14: (*химическая дезинфекция*)
Chemical(
	i_Diag:= i_DiagChemicDesinfection ,
	i_Pause:= i_Pause ,
	i_Block_Q4_in:= i_Block_Q4_in_level ,
	i_Alarm_LSmin:= i_Alarm_LSmin_Dez ,
	i_Ready_Route:= i_Ready_Route ,
	i_FS:= i_FS ,
	i_LSL:= i_LSL ,
	i_LSM:= i_LSM ,
	i_LSH:= i_LSH ,
	i_TE1:= i_TE1 ,
	i_TE2:= i_TE2 ,
	i_Current_VolumeFC1:= Current_VolumeFC1 ,
	i_Current_VolumeFC11:= Current_VolumeFC11 ,
	i_TimeDelay:= i_TimeDelay ,
	i_Time_LSH_on:= i_Time_LSH_on ,
	i_Time_LSM_on:= i_Time_LSM_on ,
	i_Time_LSM_off:= i_Time_LSM_off ,
	i_Time_LSL_off:= i_Time_LSL_off ,
	i_TimeProcess:= i_TimeChemicDesinf ,
	i_TimeSwill:= i_TimeSwillChemic ,
	i_RouteType:= i_RouteType ,
	i_PumpCapacity:= i_PumpCapacity ,
	i_TimeDelayRetPump:= i_TimeDelayRetPump ,
	i_TimeDelayRetFlow:= i_TimeDelayRetFlow ,
	i_TimeAlarmBackFlow:= i_TimeAlarmBackFlow ,
	i_VolumeDesinf:= i_VolumeDesinf ,
	q_VA541=> 	w_qDevice.VA541 ,
	q_VA401=> 	w_qDevice.VA401 ,
	q_VA11=> 	w_qDevice.VA11 ,
	q_VA551=> 	w_qDevice.VA5 ,
	q_VA501=> 	w_qDevice.VA501 ,
	q_VA51=> 	w_qDevice.VA51 ,
	q_VA511=> 	w_qDevice.VA511 ,
	q_VA521=> 	w_qDevice.VA521 ,
	q_VA531=> 	w_qDevice.VA531 ,
	q_VE551=> 	w_qDevice.VE551 ,
	q_P1=> 	w_qDevice.P1 ,
	q_P12=> q_P10 ,
	q_Red=> q_Red ,
	q_Yellow=> q_Yellow ,
	q_Green=> q_Green ,
	q_Sirena=> q_Sirena ,
	q_BackPump=> w_qDevice.BackPump ,
	q_Heating_VR1=> w_qDevice.Heating_VR1 ,
	q_AlarmBackFlow=> q_AlarmBackFlow ,
	q_Alarm_Empty_Q5=> q_Alarm_Empty_Q5 ,
	q_Vis_tim_Process=> q_Vis_tim_Process ,
	q_FC1_start=> FC1_start ,
	q_FC11_start=> FC11_start ,
	q_ZeroCount_FC1=> ZeroCount_FC1 ,
	q_ZeroCount_FC11=> ZeroCount_FC11 ,
	q_SP_P1=> q_SP_P1 ,
	q_SP_VR1=> q_SP_VR1 ,
	q_VisuMode=> q_VisuMode );
  q_Last_Time_min:=Chemical.Last_Time_min;
  q_Last_Time_sec:=Chemical.Last_Time_sec;

 T_Control_TE.IN:=w_qDevice.Heating_VR1 AND (i_TE1<(q_SP_VR1-2.0));
 T_Control_QE.IN:=Chemical.q_P12;
 q_Run_Process := (Chemical.Step < 12); (*идет подача моющих в маршрут - сигнал в маршрут*)

  IF Chemical.Step=12 THEN
     Step:=15;
  END_IF;


15: (*проверка на термическую дезинфекцию*)
 IF i_ch_ThermDesinfection THEN
    Wash_Water.Step:=0;
    Step:=16;
 ELSE
    Step:=17;
 END_IF;

16: (*термическая дезинфекция*)
Wash_Water(
	i_Diag:=i_DiagThermDesinfection ,
	i_Pause:=i_Pause ,
	i_Block_Q4_out:=i_Block_Q4_out ,
	i_Block_Q4_in:=i_Block_Q4_in_level ,
      i_Ready_Route := i_Ready_Route ,
	i_type:=1 ,
	i_FS:=i_FS ,
	i_LSL:=i_LSL ,
	i_LSM:=i_LSM ,
	i_LSH:=i_LSH ,
	i_TE1:=i_TE1 ,
	i_TE2:=i_TE2 ,
	i_Current_VolumeFC1:=Current_VolumeFC1 ,
	i_Current_VolumeFC11:=Current_VolumeFC11 ,
	i_TimeDelay:=i_TimeDelay ,
	i_Time_LSH_on:=i_Time_LSH_on ,
	i_Time_LSM_on:=i_Time_LSM_on ,
	i_Time_LSM_off:=i_Time_LSM_off ,
	i_Time_LSL_off:=i_Time_LSL_off ,
	i_TimeProcess:=i_TimeThermDesinf ,
	i_TempProcess:=i_TempThermDesinf ,
	i_DeltaTempStartTime:=i_DeltaTempStartTime ,
	i_TempCool:=i_TempCoolThermDesinf ,
	i_RouteType:=i_RouteType ,
	i_PumpCapacity:=i_PumpCapacity ,
	i_TimeDelayRetPump:=i_TimeDelayRetPump ,
	i_TimeDelayRetFlow:=i_TimeDelayRetFlow ,
	i_TimeAlarmBackFlow:=i_TimeAlarmBackFlow ,
	i_VolumeDesinf:=i_VolumeDesinf ,
	q_VA541=>	w_qDevice.VA541 ,
	q_VA401=>	w_qDevice.VA401 ,
	q_VA11=>	w_qDevice.VA11 ,
	q_VA551=>	w_qDevice.VA5 ,
	q_VA501=>	w_qDevice.VA501 ,
	q_VA51=>	w_qDevice.VA51 ,
	q_VA511=>	w_qDevice.VA511 ,
	q_VA521=>	w_qDevice.VA521 ,
	q_VA531=>	w_qDevice.VA531 ,
	q_VE551=>	w_qDevice.VE551 ,
	q_P1=>		w_qDevice.P1 ,
	q_P12=>q_P10 ,
	q_Red=>q_Red ,
	q_Yellow=>q_Yellow ,
	q_Green=>q_Green ,
	q_Sirena=>q_Sirena ,
	q_BackPump=>w_qDevice.BackPump ,
	q_Heating_VR1=>w_qDevice.Heating_VR1 ,
	q_AlarmBackFlow=>q_AlarmBackFlow ,
      q_Alarm_Empty_Q5=>q_Alarm_Empty_Q5 ,
	q_Vis_tim_Process=>q_Vis_tim_Process ,
	q_FC1_start=>FC1_start ,
	q_FC11_start=>FC11_start ,
	q_ZeroCount_FC1=>ZeroCount_FC1 ,
	q_ZeroCount_FC11=>ZeroCount_FC11 ,
	q_SP_P1=>q_SP_P1 ,
	q_SP_VR1=>q_SP_VR1 ,
	q_VisuMode=>q_VisuMode );
  q_Last_Time_min:=Wash_Water.Last_Time_min;
  q_Last_Time_sec:=Wash_Water.Last_Time_sec;

 T_Control_TE.IN:=w_qDevice.Heating_VR1 AND (i_TE1<(q_SP_VR1-2.0));
 q_Run_Process := (Wash_Water.Step<9); (*идет подача моющих в маршрут - сигнал в маршрут*)

  IF Wash_Water.Step=10 THEN
     Step:=17;
  END_IF;

17: (*автоматическая мойка закончена*)
    T_Imp_EndAutoMode.IN := TRUE;
    Step:=0;

18: (*ручной режим*)
Hand_Mode(
	i_Diag:=			i_DiagHandMode ,
	i_Alarm_PE:=	i_Alarm_PE ,
	Man_VA541:=		w_ManDevice.VA541,
	Man_VA401:=		w_ManDevice.VA401,
	Man_VA201:=		w_ManDevice.VA201,
	Man_VA301:=		w_ManDevice.VA301,
	Man_VA41:=			w_ManDevice.VA41,
	Man_VA11:=			w_ManDevice.VA11,
	Man_VA21:=			w_ManDevice.VA21,
	Man_VA31:=			w_ManDevice.VA31,
	Man_VA5:=			w_ManDevice.VA5,
	Man_VA501:=		w_ManDevice.VA501,
	Man_VA51:=			w_ManDevice.VA51,
	Man_VA511:=		w_ManDevice.VA511,
	Man_VA521:=		w_ManDevice.VA521,
	Man_VA531:=		w_ManDevice.VA531,
	Man_P1:=			w_ManDevice.P1,
	Man_BackPump:=	w_ManDevice.BackPump,
	Man_VR1:=			w_ManDevice.Heating_VR1,
	Man_VE551:=		w_ManDevice.VE551,
	Man_ZeroCount_FC1:=w_ManDevice.Zero_FC1,
	Man_ZeroCount_FC11:=	w_ManDevice.Zero_FC11,
	Man_VE7:=		Man_VE7,
	Man_P8:=		Man_P8,
	Man_P9:=		Man_P9,
	Man_P10:=		Man_P10,
	ManSP_P1:=	ManSP_P1,
	ManSP_VR1	:=	ManSP_VR1,
	q_VA541=>	w_qDevice.VA541 ,
	q_VA401=>	w_qDevice.VA401 ,
	q_VA201=>	w_qDevice.VA201 ,
	q_VA301=>	w_qDevice.VA301 ,
	q_VA41=>	w_qDevice.VA41 ,
	q_VA11=>	w_qDevice.VA11 ,
	q_VA21=>	w_qDevice.VA21 ,
	q_VA31=>	w_qDevice.VA31 ,
	q_VA5=>	w_qDevice.VA5 ,
	q_VA501=>	w_qDevice.VA501 ,
	q_VA51=>	w_qDevice.VA51 ,
	q_VA511=>	w_qDevice.VA511 ,
	q_VA521=>	w_qDevice.VA521 ,
	q_VA531=>	w_qDevice.VA531 ,
	q_P1=>		w_qDevice.P1 ,
	q_BackPump=>	w_qDevice.BackPump ,
	q_Heating_VR1=>	w_qDevice.Heating_VR1 ,
	q_VE551=>	w_qDevice.VE551 ,
	q_VE7=>q_VE7 ,
	q_P8=>q_P8 ,
	q_P9=>q_P9 ,
	q_P10=>q_P10 ,
	q_Red=>q_Red ,
	q_Yellow=>q_Yellow ,
	q_Green=>q_Green ,
	q_Sirena=>q_Sirena ,
	q_FC1_start=>FC1_start ,
	q_FC11_start=>FC11_start ,
	q_ZeroCount_FC1=>ZeroCount_FC1 ,
	q_ZeroCount_FC11=>ZeroCount_FC11 ,
	q_SP_P1=>q_SP_P1 ,
	q_SP_VR1=>q_SP_VR1 ,
	q_VisuMode=>q_VisuMode ,
	q_ModeQE=>q_ModeQE);

19: (*подготовка щелочи*)
    q_ModeQE:=0;  (*режим выбора пересчета концентрации*)
    q_Block_Solution_Alk:=TRUE;
Preparation(
	i_Diag:=i_DiagPrepareAlkaline ,
	i_Pause:=i_Pause ,
	i_Block_Q4_out:=i_Block_Q4_out ,
	i_Block_Q4_in:=i_Block_Q4_in_level AND i_Block_Q4_in_ph ,
	i_Alarm_LSmin:=i_Alarm_LSmin_Alk ,
    i_Alk:=TRUE,
	i_FS:=i_FS ,
	i_TE1:=i_TE1 ,
	i_TE2:=i_TE2 ,
	i_TE_tank:=i_TE_Q2 ,
	i_LE_tank:=i_LE_Q2 ,
	i_QE:=i_QE ,
	i_QE_priv:=i_QE_priv ,
	i_TimeDelay:=i_TimeDelay ,
	i_MaxCondPrep:=MaxCondPrepAlk ,
	i_MinCondPrep:=MinCondPrepAlk ,
	i_MaxTempPrep:=MaxTempPrepAlk ,
	i_MinTempPrep:=MinTempPrepAlk ,
	i_LvlPrep:=LvlPrepAlk ,
	q_VA541=>	w_qDevice.VA541 ,
	q_VA401=>	w_qDevice.VA401 ,
	q_VA201=>	w_qDevice.VA201 ,
	q_VA41=>	w_qDevice.VA41 ,
	q_VA11=>	w_qDevice.VA11 ,
	q_VA21=>	w_qDevice.VA21 ,
	q_VA551=>	w_qDevice.VA5 ,
	q_VA501=>	w_qDevice.VA501 ,
	q_VA51=>	w_qDevice.VA51 ,
	q_VA511=>	w_qDevice.VA511 ,
	q_VA521=>	w_qDevice.VA521 ,
	q_VA531=>	w_qDevice.VA531 ,
	q_VE11=>q_VE7 ,
	q_P1=>		w_qDevice.P1 ,
	q_P10=>q_P9 ,
	q_Red=>q_Red ,
	q_Yellow=>q_Yellow ,
	q_Green=>q_Green ,
	q_Sirena=>q_Sirena ,
	q_Heating_VR1=>	w_qDevice.Heating_VR1 ,
	q_AlarmBackFlow=>q_AlarmBackFlow ,
	q_Vis_tim_Process=>q_Vis_tim_Process ,
	q_SP_P1=>q_SP_P1 ,
	q_SP_VR1=>q_SP_VR1 ,
	q_VisuMode=>q_VisuMode );
  q_Last_Time_min:=Preparation.Last_Time_min;
  q_Last_Time_sec:=Preparation.Last_Time_sec;

 T_Control_TE.IN:=w_qDevice.Heating_VR1 AND (i_TE1<(q_SP_VR1-2.0));
 T_Control_QE.IN:=Preparation.q_P10;

  IF Preparation.Step=12 THEN
     Step:=0;
  END_IF;

20: (*подготовка кислоты*)
    q_ModeQE:=1;  (*режим выбора пересчета концентрации*)
    q_Block_Solution_Acid:=TRUE;
Preparation(
	i_Diag:=i_DiagPrepareAcid ,
	i_Pause:=i_Pause ,
	i_Block_Q4_out:=i_Block_Q4_out ,
	i_Block_Q4_in:=i_Block_Q4_in_level AND i_Block_Q4_in_ph ,
	i_Alarm_LSmin:=i_Alarm_LSmin_Acid ,
    i_Alk:=FALSE,
	i_FS:=i_FS ,
	i_TE1:=i_TE1 ,
	i_TE2:=i_TE2 ,
	i_TE_tank:=i_TE_Q3 ,
	i_LE_tank:=i_LE_Q3 ,
	i_QE:=i_QE ,
	i_QE_priv:=i_QE_priv ,
	i_TimeDelay:=i_TimeDelay ,
	i_MaxCondPrep:=MaxCondPrepAcid ,
	i_MinCondPrep:=MinCondPrepAcid ,
	i_MaxTempPrep:=MaxTempPrepAcid ,
	i_MinTempPrep:=MinTempPrepAcid ,
	i_LvlPrep:=LvlPrepAcid ,
	q_VA541=>	w_qDevice.VA541 ,
	q_VA401=>	w_qDevice.VA401 ,
	q_VA201=>	w_qDevice.VA301 ,
	q_VA41=>	w_qDevice.VA41 ,
	q_VA11=>	w_qDevice.VA11 ,
	q_VA21=>	w_qDevice.VA31 ,
	q_VA551=>	w_qDevice.VA5 ,
	q_VA501=>	w_qDevice.VA501 ,
	q_VA51=>	w_qDevice.VA51 ,
	q_VA511=>	w_qDevice.VA511 ,
	q_VA521=>	w_qDevice.VA521 ,
	q_VA531=>	w_qDevice.VA531 ,
	q_VE11=>q_VE7 ,
	q_P1=>		w_qDevice.P1 ,
	q_P10=>q_P8 ,
	q_Red=>q_Red ,
	q_Yellow=>q_Yellow ,
	q_Green=>q_Green ,
	q_Sirena=>q_Sirena ,
	q_Heating_VR1=>	w_qDevice.Heating_VR1 ,
	q_AlarmBackFlow=>q_AlarmBackFlow ,
	q_Vis_tim_Process=>q_Vis_tim_Process ,
	q_SP_P1=>q_SP_P1 ,
	q_SP_VR1=>q_SP_VR1 ,
	q_VisuMode=>q_VisuMode );
  q_Last_Time_min:=Preparation.Last_Time_min;
  q_Last_Time_sec:=Preparation.Last_Time_sec;

 T_Control_TE.IN:=w_qDevice.Heating_VR1 AND (i_TE1<(q_SP_VR1-2.0));
 T_Control_QE.IN:=Preparation.q_P10;

  IF Preparation.Step=12 THEN
     Step:=0;
  END_IF;

21: (*диагностика*)
Diagn(
	i_Diag:=i_DiagDiagnostic ,
	q_VA541=>	w_qDevice.VA541 ,
	q_VA401=>	w_qDevice.VA401 ,
	q_VA201=>	w_qDevice.VA201 ,
	q_VA301=>	w_qDevice.VA301 ,
	q_VA41=>	w_qDevice.VA41 ,
	q_VA11=>	w_qDevice.VA11 ,
	q_VA21=>	w_qDevice.VA21 ,
	q_VA31=>	w_qDevice.VA31 ,
	q_VA551=>	w_qDevice.VA5 ,
	q_VA501=>	w_qDevice.VA501 ,
	q_VA51=>	w_qDevice.VA51 ,
	q_VA511=>	w_qDevice.VA511 ,
	q_VA521=>	w_qDevice.VA521 ,
	q_VA531=>	w_qDevice.VA531 ,
	q_Red=>q_Red ,
	q_Yellow=>q_Yellow ,
	q_Green=>q_Green ,
	q_Sirena=>q_Sirena ,
	q_VisuMode=>q_VisuMode );

  IF Diagn.Step=15 THEN
     Step:=0;
  END_IF;

END_CASE;




(*работа расходомера дезинфектанта*)
fp_FC1_imp(CLK:=i_FS1 ); (*передний фронт импульса*)
IF FC1_start THEN
 IF fp_FC1_imp.Q THEN
    Current_VolumeFC1:=Current_VolumeFC1+i_K_imp_dez;
 END_IF;
END_IF;
IF ZeroCount_FC1 THEN  (*обнуление счетчика*)
   Current_VolumeFC1:=0.0;
END_IF;
(*работа расходомера подачи*)
fp_FC11_imp(CLK:=i_FC11 ); (*передний фронт импульса*)
IF FC11_start THEN
 IF fp_FC11_imp.Q THEN
    Current_VolumeFC11:=Current_VolumeFC11+i_K_imp;
 END_IF;
END_IF;
IF ZeroCount_FC11 THEN  (*обнуление счетчика*)
   Current_VolumeFC11:=0.0;
END_IF;



IF AlarmReset AND T_Control_TE.Q THEN
 T_Control_TE.IN:=FALSE;
END_IF;
IF AlarmReset AND T_Control_QE.Q THEN
 T_Control_QE.IN:=FALSE;
END_IF;

T_Control_TE(PT:=DINT_TO_TIME(Time_Control_TE*60000)); (*таймер контроля набора температуры*)
T_Control_QE(PT:=DINT_TO_TIME(Time_Control_QE*60000)); (*таймер контроля набора концентрации*)
T_Imp_EndAutoMode(PT:=T#7s , Q=>q_End_AutoMode );  (*импульсный таймер выдачи сигнала "мойка закончена" в маршрут*)
END_FUNCTION_BLOCK

(* POU SolutionPrepar, ST *)
FUNCTION_BLOCK SolutionPrepar
VAR_INPUT
	i_Diag			: BOOL;
	i_Pause			: BOOL;
	i_Block_Q4_out  	: BOOL; 	(*блокировка выпуска для полоскания из Q4  - мин уровень и ph*)
	i_Block_Q4_in   	: BOOL; 	(*блокировка подачи в Q4 - макс уровень и ph*)
	i_Alarm_LSmin	: BOOL;   	(*авария нижнего уровня в баке концентрата*)
	i_Alk			: BOOL;       (*подготовка щелочи*)
	i_FS			: BOOL;       (*датчик протока на возврате*)

	i_TE1			: REAL;      	(*температура на подаче*)
	i_TE2			: REAL;      	(*температура на возврате*)
	i_TE_tank		: REAL;  	(*температура в танке раствора*)
	i_LE_tank		: REAL;  	(*уровень в танке раствора*)
	i_QE 			: REAL;      	(*расчитанная концентрация % раствора*)
	i_QE_priv 		: REAL; 		(*приведенная проводимость к температуре*)

	i_TimeDelay    	: DINT ; 		(*время задержки вкл/выкл клапанов и насосов*)

	i_MaxCondPrep	: REAL;  	(*максимальная проводимость раствора при подготовке*)
	i_MinCondPrep	: REAL;  	(*минимальная проводимость раствора при подготовке*)
	i_MaxTempPrep	: REAL;  	(*максимальная темп при подготовке*)
	i_MinTempPrep	: REAL;  	(*минимальная темп при подготовке*)
	i_LvlPrep		: INT;       	(*заданный уровень в баке раствора при подготовке*)

    	Step	: INT;
END_VAR
VAR_OUTPUT
	q_VA541	: BOOL;
	q_VA401	: BOOL;
	q_VA201	: BOOL;
	q_VA41 		: BOOL;
	q_VA11 		: BOOL;
	q_VA21 		: BOOL;
	q_VA551	: BOOL;
	q_VA501	: BOOL;
	q_VA51 		: BOOL;
	q_VA511	: BOOL;
	q_VA521	: BOOL;
	q_VA531	: BOOL;
	q_VE11 		: BOOL;
	q_P1   		: BOOL;
	q_P10  		: BOOL;
	q_Red  		: BOOL;
	q_Yellow 	: BOOL;
	q_Green  	: BOOL;
	q_Sirena 	: BOOL;
	q_Heating_VR1		: BOOL;
	q_AlarmBackFlow	: BOOL;  (* авария протока на возврате*)
	q_Vis_tim_Process	: BOOL;
	q_SP_P1 			: REAL;
	q_SP_VR1			: REAL;
	q_VisuMode			: INT;
END_VAR

VAR

	EjectionAlk        	AT %M*: BOOL; 		(*была подача щелочи,необходимость промывки линии*)
	PastPrev           	AT %M*: INT;
	Last_Time_min  	AT %M*: DINT;  		(*расчет оставшихся минут процесса*)
	Last_Time_sec  	AT %M*: DINT;  		(*расчет оставшихся секунд процесса*)

	T_Delay   	:TON;  (*служебный таймер*)
	T_Process 	:TON;
END_VAR
(*обнуление в начале скана*)
	q_VA541 := FALSE;  (*НО*)
	q_VA401 := FALSE;
	q_VA201 := FALSE;
	q_VA41  := FALSE;
	q_VA11  := FALSE;
	q_VA21  := FALSE;
	q_VA551 := FALSE;
	q_VA501 := FALSE;
	q_VA51  := FALSE;
	q_VA511 := FALSE;
	q_VA521 := FALSE;
	q_VA531 := FALSE;  (*НО*)
	q_VE11  := FALSE;
	q_P1 := FALSE;
	q_P10 := FALSE;
    q_Green :=FALSE;
    q_Yellow :=FALSE;
    q_Red:=FALSE;
    q_Sirena :=FALSE;
    q_Heating_VR1 := FALSE;
    q_AlarmBackFlow := FALSE;
    q_Vis_tim_Process:=FALSE;
	q_SP_P1 :=0.0 ;
	q_SP_VR1 :=0.0 ;

(*выход в аварию*)
IF i_Diag   THEN
   IF Step=0 THEN
      PastPrev:=0;
   END_IF;
   Step:=30;
END_IF;

(*выход в паузу*)
IF i_Pause   THEN
   IF Step=0 THEN
      PastPrev:=0;
   END_IF;
   Step:=35;
END_IF;

CASE Step OF
0: (*обнуление*)
  EjectionAlk:=FALSE;
  T_Delay.IN:=FALSE;
  T_Process.IN:=FALSE;
  Step:=1;

1: (*проверка уровня*)
  IF i_LE_tank<i_LvlPrep THEN
    Step:=2;
  ELSE
    Step:=4 ;
  END_IF;

2: (*пополнение танка водой*)
  PastPrev:=Step;
  q_VA11:=TRUE;
  q_VA521:=TRUE;
  q_VA531:=TRUE;
  q_VA541:=TRUE;
  q_VA201:=TRUE;
  q_P1:=TRUE;
  q_SP_P1:=FlowPrep;

     (*нагрев*)
     IF i_TE_tank<i_MaxTempPrep THEN
        q_Heating_VR1:=TRUE;
        q_SP_VR1:=i_MaxTempPrep+10.0;
     END_IF;

  T_Delay.PT:=DINT_TO_TIME(i_TimeDelay*1000);
  T_Delay.IN:=i_LE_tank>i_LvlPrep;
  IF T_Delay.Q THEN
     T_Delay.IN:=FALSE;
     Step:=3;
  END_IF;

  q_VisuMode:=5;

3: (*переключение*)
  PastPrev:=Step;
  q_VA11:=TRUE;
  q_VA21:=TRUE;
  q_VA521:=TRUE;
  q_VA531:=TRUE;
  q_VA541:=TRUE;
  q_VA201:=TRUE;
  q_P1:=TRUE;
  q_SP_P1:=FlowPrep;

     (*нагрев*)
     IF i_TE_tank<i_MaxTempPrep THEN
        q_Heating_VR1:=TRUE;
        q_SP_VR1:=i_MaxTempPrep+10.0;
     END_IF;

  T_Delay.PT:=DINT_TO_TIME(i_TimeDelay*1000);
  T_Delay.IN:=TRUE;
  IF T_Delay.Q THEN
     T_Delay.IN:=FALSE;
     Step:=4;
  END_IF;

  q_VisuMode:=5;

4: (*перемешивание*)
  PastPrev:=Step;
  q_VA21:=TRUE;
  q_VA521:=TRUE;
  q_VA531:=TRUE;
  q_VA541:=TRUE;
  q_VA201:=TRUE;
  q_P1:=TRUE;
  q_SP_P1:=FlowPrep;
     (*нагрев*)
     IF i_TE_tank<i_MaxTempPrep THEN
        q_Heating_VR1:=TRUE;
        q_SP_VR1:=i_MaxTempPrep+10.0;
     END_IF;

   (*вытеснение концентрата щелочи*)
  IF T_Process.ET<DINT_TO_TIME(EjectTime*1000) THEN
     q_P10:=EjectionAlk ;
     q_VE11:=EjectionAlk;
  END_IF;

     (*расчет времени для визуализ*)
    q_Vis_tim_Process := TRUE; (*визуализация полей времени*)
    Last_Time_min := (TIME_TO_DINT(T_Process.PT-T_Process.ET))/60000 ;
    Last_Time_sec := (TIME_TO_DINT(T_Process.PT-T_Process.ET)/1000) - Last_Time_min * 60 ;

   T_Process.PT:=DINT_TO_TIME(TimeMixPrep*1000);
   T_Process.in:=TRUE;
   IF T_Process.q AND i_QE<i_MaxCondPrep THEN
      T_Process.in:=FALSE;
      EjectionAlk:=FALSE;
      Step:=5;
   ELSIF T_Process.q AND i_QE>=i_MaxCondPrep THEN
      T_Process.in:=FALSE;
      EjectionAlk:=FALSE;
      Step:=6;
   END_IF;

  q_VisuMode:=6;

5: (*набор концентрации*)
  PastPrev:=Step;
  q_VA21:=TRUE;
  q_VA521:=TRUE;
  q_VA531:=TRUE;
  q_VA541:=TRUE;
  q_VA201:=TRUE;
  q_P1:=TRUE;
  q_SP_P1:=FlowPrep;
     (*нагрев*)
     IF i_TE_tank<i_MaxTempPrep THEN
        q_Heating_VR1:=TRUE;
        q_SP_VR1:=i_MaxTempPrep+10.0;
     END_IF;

  q_P10:=TRUE;
  EjectionAlk:=i_Alk;

   IF i_QE>=i_MaxCondPrep THEN
      T_Process.in:=FALSE;
      Step:=4;
   END_IF;
   IF i_Alarm_LSmin THEN  (*мин уровень в баке концентрата*)
      Step:=30;
   END_IF;

  q_VisuMode:=7;

6: (*догрев*)
  PastPrev:=Step;
  q_VA21:=TRUE;
  q_VA521:=TRUE;
  q_VA531:=TRUE;
  q_VA541:=TRUE;
  q_VA201:=TRUE;
  q_P1:=TRUE;
  q_SP_P1:=FlowPrep;
  q_Heating_VR1:=TRUE;
  q_SP_VR1:=i_MaxTempPrep+10.0;

  IF i_TE_tank>=i_MaxTempPrep THEN
     Step:=7;
  END_IF;

  q_VisuMode:=8;

7: (*переключение*)
  PastPrev:=Step;
  q_VA11:=TRUE;
  q_VA21:=TRUE;
  q_VA521:=TRUE;
  q_VA531:=TRUE;
  q_VA541:=TRUE;
  q_VA201:=TRUE;
  q_P1:=TRUE;
  q_SP_P1:=FlowPrep;

  T_Delay.PT:=DINT_TO_TIME(i_TimeDelay*1000);
  T_Delay.IN:=TRUE;
  IF T_Delay.Q THEN
     T_Delay.IN:=FALSE;
     Step:=8;
  END_IF;

  q_VisuMode:=1;

8: (*вытеснение в танк раствора*)
  PastPrev:=Step;
  q_VA11:=TRUE;
  q_VA521:=TRUE;
  q_VA531:=TRUE;
  q_VA541:=TRUE;
  q_VA201:=TRUE;
  q_P1:=TRUE;
  q_SP_P1:=FlowPrep;

  IF i_QE<i_MaxCondPrep/3 THEN
     Step:=9;
  END_IF;

  q_VisuMode:=1;

9: (*переключение*)
  PastPrev:=Step;
  q_VA11:=TRUE;
  q_VA521:=TRUE;
  q_VA531:=TRUE;
  q_VA541:=TRUE;
  q_VA201:=TRUE;
  q_VA401:=TRUE;
  q_P1:=TRUE;
  q_SP_P1:=FlowPrep;

  T_Delay.PT:=DINT_TO_TIME(i_TimeDelay*1000);
  T_Delay.IN:=TRUE;
  IF T_Delay.Q THEN
     T_Delay.IN:=FALSE;
     Step:=10;
  END_IF;

  q_VisuMode:=1;

10: (*вытеснение в танк Q4*)
  PastPrev:=Step;
  q_VA11:=TRUE;
  q_VA521:=TRUE;
  q_VA531:=TRUE;
  q_VA541:=TRUE;
  q_VA401:=TRUE;
  q_P1:=TRUE;
  q_SP_P1:=FlowPrep;

  IF i_QE_priv<5.0 THEN
     Step:=11;
  END_IF;

  q_VisuMode:=1;

11: (*переключение*)
  PastPrev:=Step;
  q_VA11:=TRUE;
  q_VA521:=TRUE;
  q_VA531:=TRUE;
  q_VA541:=TRUE;
  q_VA401:=TRUE;

  T_Delay.PT:=T#5s;
  T_Delay.IN:=TRUE;
  IF T_Delay.Q THEN
     T_Delay.IN:=FALSE;
     Step:=12;
  END_IF;

  q_VisuMode:=1;

12: (*остановка*)
  q_VisuMode:=1;




(*-----------------авария----------------*)
30: (*авария*)
       q_VisuMode:=11;
       q_Red:=TRUE;
       q_Sirena :=TRUE;
       T_Process.IN := FALSE; (*остановка таймера процесса*)
       IF  AlarmReset THEN
          Step := PastPrev;
       END_IF;

(*-----------------пауза----------------*)
35: (*пауза*)
       q_VisuMode:=12;
       q_Yellow:=TRUE;
       T_Process.IN := FALSE; (*остановка таймера процесса*)
       IF NOT i_Pause  THEN
          Step := PastPrev;
       END_IF;
 END_CASE;

T_Delay();
T_Process();
END_FUNCTION_BLOCK

(* POU Manual, ST *)
FUNCTION_BLOCK Manual
VAR_INPUT
	i_Diag		: BOOL;
	i_Alarm_PE	: BOOL;    (*Превышение давления в контуре*)

    Step: INT;

(*команды ручного режима контура*)
	Man_VA541   			: BOOL;		(*VA541 Клапан сброса в канализацию из контура *)
	Man_VA401    			: BOOL;		(*VA401 Клапан подачи в бак возвратной воды *)
	Man_VA201    			: BOOL;		(*VA201 Клапан подачи в бак щелочи *)
	Man_VA301    			: BOOL;		(*VA301 Клапан подачи в бак кислоты *)
	Man_VA41     			: BOOL;		(*VA41 Клапан выпуска из бака возвратной воды*)
	Man_VA11     			: BOOL;		(*VA11 Клапан выпуска из бака чистой воды*)
	Man_VA21     			: BOOL;		(*VA21 Клапан выпуска из бака щелочи*)
	Man_VA31     			: BOOL;		(*VA31 Клапан выпуска из бака кислоты*)
	Man_VA5    				: BOOL;		(*VA5 Клапан подачи чистой воды в цирк бак*)
	Man_VA501    			: BOOL;		(*VA501 Клапан подачи растворов в цирк бак*)
	Man_VA51     			: BOOL;		(*VA51  Клапан выпуска из цирк бака*)
	Man_VA511    			: BOOL;		(*VA511 Клапан выпуска в канализацию из цирк бака*)
	Man_VA521    			: BOOL;		(*VA521 Клапан циркуляции по контуру*)
	Man_VA531    			: BOOL;		(*VA531 Клапан подачи из контура в маршрут*)
	Man_P1       				: BOOL;		(*Р1 Старт насоса подачи *)
	Man_BackPump 			: BOOL;		(*Старт насоса возврата*)
	Man_VR1      			: BOOL;		(*Включение нагрева*)
	Man_VE551    			: BOOL;		(*VE551 Клапан дезинфектанта*)

(*команды ручного режима общих механизмов*)
	Man_VE7     			: BOOL;		(*VE7 Клапан промывки линии концентрата щелочи*)
	Man_P8      				: BOOL;		(*Р8 Насос-дозатор концентрата  кислоты*)
	Man_P9      				: BOOL;		(*Р9 Насос-дозатор концентрата  щелочи*)
	Man_P10      			: BOOL;		(*Р10 Насос-дозатор дезинфектанта*)

	Man_ZeroCount_FC1 	: BOOL;		(*Обнуление расходомера подачи*)
	Man_ZeroCount_FC11 	: BOOL;		(*Обнуление расходомера дезинфектанта*)

	ManSP_P1    	 		: REAL;		(*задание производительности насоса подачи в ручном режиме*)
	ManSP_VR1    			: REAL;		(*задание температуры нагрева в ручном режиме*)

END_VAR

VAR_OUTPUT
	q_VA541		: BOOL;		(*VA541 Клапан сброса в канализацию из контура *)
	q_VA401		: BOOL;		(*VA401 Клапан подачи в бак возвратной воды *)
	q_VA201		: BOOL;		(*VA201 Клапан подачи в бак щелочи *)
	q_VA301		: BOOL;		(*VA301 Клапан подачи в бак кислоты *)
	q_VA41 			: BOOL;		(*VA41 Клапан выпуска из бака возвратной воды*)
	q_VA11 			: BOOL;		(*VA11 Клапан выпуска из бака чистой воды*)
	q_VA21 			: BOOL;		(*VA21 Клапан выпуска из бака щелочи*)
	q_VA31 			: BOOL;		(*VA31 Клапан выпуска из бака кислоты*)
	q_VA5			: BOOL;		(*VA5 Клапан подачи чистой воды в цирк бак*)
	q_VA501		: BOOL;		(*VA501 Клапан подачи растворов в цирк бак*)
	q_VA51 			: BOOL;		(*VA51  Клапан выпуска из цирк бака*)
	q_VA511		: BOOL;		(*VA511 Клапан выпуска в канализацию из цирк бака*)
	q_VA521		: BOOL;		(*VA521 Клапан циркуляции по контуру*)
	q_VA531		: BOOL;		(*VA531 Клапан подачи из контура в маршрут*)
	q_P1   			: BOOL;		(*Р1 Старт насоса подачи *)
	q_BackPump	: BOOL;		(*Старт насоса возврата*)
	q_Heating_VR1	: BOOL;		(*Включение нагрева*)
	q_VE551		: BOOL;		(*VE551 Клапан дезинфектанта*)

	q_VE7 			: BOOL;		(*VE7 Клапан промывки линии концентрата щелочи*)
	q_P8  			: BOOL;		(*Р8 Насос-дозатор концентрата  кислоты*)
	q_P9  			: BOOL;		(*Р9 Насос-дозатор концентрата  щелочи*)
	q_P10  			: BOOL;		(*Р10 Насос-дозатор дезинфектанта*)

	q_Red  			: BOOL;		(*Светозвуковая сигнализация. Красный свет*)
	q_Yellow 		: BOOL;		(*Светозвуковая сигнализация. Желтый свет*)
	q_Green  		: BOOL;		(*Светозвуковая сигнализация. Зеленый свет*)
	q_Sirena 		: BOOL;		(*Светозвуковая сигнализация. Зуммер*)


	q_FC1_start 			: BOOL;   	(*старт подсчета импульсов дезинф*)
	q_FC11_start		: BOOL;	  	(*старт подсчета импульсов*)
	q_ZeroCount_FC1	: BOOL; 	(*обнуление счетчика дезинф*)
	q_ZeroCount_FC11	: BOOL; 	(*обнуление счетчика*)

	q_SP_P1 		: REAL;		(*задание производительности насоса подачи в ручном режиме*)
	q_SP_VR1		: REAL;		(*задание температуры нагрева в ручном режиме*)

	q_VisuMode		: INT;
	q_ModeQE 		: INT;     		(*режим выбора пересчета концентрации, 0-щелочь, 1-кислота*)
END_VAR

VAR

END_VAR
(*обнуление в начале скана*)
	q_VA541 := FALSE;
	q_VA401 := FALSE;
	q_VA201 := FALSE;
	q_VA301 := FALSE;
	q_VA41  := FALSE;
	q_VA11  := FALSE;
	q_VA21  := FALSE;
	q_VA31  := FALSE;
	q_VA5    := FALSE;
	q_VA501 := FALSE;
	q_VA51  := FALSE;
	q_VA511 := FALSE;
	q_VA521 := FALSE;
	q_VA531 := FALSE;
	q_P1 := FALSE;
	q_BackPump := FALSE;
   	q_Heating_VR1 := FALSE;
	q_VE551 := FALSE;
	q_ZeroCount_FC1  := FALSE;
	q_ZeroCount_FC11 := FALSE;

	q_VE7  := FALSE;
	q_P8 := FALSE;
	q_P9 := FALSE;
	q_P10 := FALSE;

    	q_Green :=FALSE;
    	q_Yellow :=FALSE;
    	q_Red:=FALSE;
    	q_Sirena :=FALSE;

	q_FC1_start  := FALSE;
	q_FC11_start := FALSE;

	q_SP_P1 :=0.0 ;
	q_SP_VR1 :=0.0 ;

(*выход в аварию*)
 IF i_Diag   THEN
   Step:=30;
END_IF;


CASE Step OF
0: (*обнуление*)
	Man_VA541  :=FALSE;
	Man_VA401  :=FALSE;
	Man_VA201  :=FALSE;
	Man_VA301  :=FALSE;
	Man_VA41    :=FALSE;
	Man_VA11    :=FALSE;
	Man_VA21    :=FALSE;
	Man_VA31    :=FALSE;
	Man_VA5      :=FALSE;
	Man_VA501  :=FALSE;
	Man_VA51    :=FALSE;
	Man_VA511  :=FALSE;
	Man_VA521  :=FALSE;
	Man_VA531  :=FALSE;
	Man_P1        :=FALSE;
	Man_BackPump:=FALSE;
	Man_VR1     :=FALSE;
	Man_VE551 :=FALSE;
	Man_ZeroCount_FC1:=FALSE;
	Man_ZeroCount_FC11:=FALSE;
	Man_VE7    :=FALSE;
	Man_P8      :=FALSE;
	Man_P9      :=FALSE;
	Man_P10    :=FALSE;

	ManSP_P1    :=0.0;
	ManSP_VR1   :=0.0;

    Step:=1;

1: (*ручной режим*)
	q_VA541 := Man_VA541;
	q_VA401 := Man_VA401;
	q_VA201 := Man_VA201;
	q_VA301 := Man_VA301;
	q_VA41  := Man_VA41;
	q_VA11  := Man_VA11;
	q_VA21  := Man_VA21;
	q_VA31  := Man_VA31;
	q_VA5 := Man_VA5;
	q_VA501 := Man_VA501;
	q_VA51  := Man_VA51;
	q_VA511 := Man_VA511;
	q_VA521 := Man_VA521;
	q_VA531 := Man_VA531;
	q_VE7  := Man_VE7;
	q_VE551 := Man_VE551;

    IF q_VA21 THEN (*режим выбора пересчета концентрации, 0-щелочь, 1-кислота*)
       q_ModeQE :=0;
    ELSIF q_VA31 THEN
       q_ModeQE :=1;
    END_IF;


    (*--------насосы-----------*)
    IF i_Alarm_PE THEN
       q_P1:=FALSE;
       q_SP_P1 := 0.0;
    ELSE
       q_P1 :=  Man_P1;
       q_SP_P1 := ManSP_P1; (*задание  на частотник насоса*)
    END_IF;

    q_P8 :=  Man_P8;
    q_P9 :=  Man_P9;
    q_P10 :=  Man_P10;

    q_BackPump:=Man_BackPump;


    (*-------аналоговые клапана-------*)
    q_Heating_VR1 := q_P1 AND Man_VR1;
    q_SP_VR1 := ManSP_VR1;


    (*--------расходомеры-------------*)
	q_FC1_start :=TRUE;
	q_FC11_start:=TRUE;
	q_ZeroCount_FC1:=Man_ZeroCount_FC1;   (*обнуление*)
	q_ZeroCount_FC11:=Man_ZeroCount_FC11; (*обнуление*)


     q_Green :=TRUE;
     q_VisuMode:=1;

30:  (*авария*)
	Man_VA541  :=FALSE;
	Man_VA401  :=FALSE;
	Man_VA201  :=FALSE;
	Man_VA301  :=FALSE;
	Man_VA41    :=FALSE;
	Man_VA11    :=FALSE;
	Man_VA21    :=FALSE;
	Man_VA31    :=FALSE;
	Man_VA5      :=FALSE;
	Man_VA501  :=FALSE;
	Man_VA51    :=FALSE;
	Man_VA511  :=FALSE;
	Man_VA521  :=FALSE;
	Man_VA531  :=FALSE;
	Man_P1        :=FALSE;
	Man_BackPump:=FALSE;
	Man_VR1     :=FALSE;
	Man_VE551 :=FALSE;
	Man_ZeroCount_FC1:=FALSE;
	Man_ZeroCount_FC11:=FALSE;
	Man_VE7    :=FALSE;
	Man_P8      :=FALSE;
	Man_P9      :=FALSE;
	Man_P10    :=FALSE;

	ManSP_P1    :=0.0;
	ManSP_VR1   :=0.0;


  IF AlarmReset THEN   (*сброс аварии*)
     Step:=1;
  END_IF;
    q_VisuMode:=11;

     q_Red:=TRUE;
     q_Sirena :=TRUE;

END_CASE;
END_FUNCTION_BLOCK

(* POU Diagnostic, ST *)
FUNCTION_BLOCK Diagnostic
VAR_INPUT
	i_Diag	: BOOL;
	Step	: INT;
END_VAR
VAR_OUTPUT
	q_VA541	: BOOL;
	q_VA401	: BOOL;
	q_VA201	: BOOL;
	q_VA301	: BOOL;
	q_VA41 		: BOOL;
	q_VA11 		: BOOL;
	q_VA21 		: BOOL;
	q_VA31 		: BOOL;
	q_VA551	: BOOL;
	q_VA501	: BOOL;
	q_VA51 		: BOOL;
	q_VA511	: BOOL;
	q_VA521	: BOOL;
	q_VA531	: BOOL;
	q_Red  		: BOOL;
	q_Yellow 	: BOOL;
	q_Green  	: BOOL;
	q_Sirena 	: BOOL;
	q_VisuMode 	: INT;
END_VAR



VAR
	PastPrev  	: INT;
	T_StepFW	:TON;
END_VAR
(*обнуление в начале скана*)
	q_VA541 := FALSE;
	q_VA401 := FALSE;
	q_VA201 := FALSE;
	q_VA301 := FALSE;
	q_VA41  := FALSE;
	q_VA11  := FALSE;
	q_VA21  := FALSE;
	q_VA31  := FALSE;
	q_VA551 := FALSE;
	q_VA501 := FALSE;
	q_VA51  := FALSE;
	q_VA511 := FALSE;
	q_VA521 := FALSE;
	q_VA531 := FALSE;
    q_Green :=FALSE;
    q_Yellow :=FALSE;
    q_Red:=FALSE;
    q_Sirena :=FALSE;

(*выход в аварию*)
IF i_Diag THEN
   IF Step=0 THEN
      PastPrev:=0;
   END_IF;
   Step:=30;
END_IF;

q_VisuMode:=1;

CASE Step OF
0: (*обнуление*)
   T_StepFW.IN := FALSE;
   Step:=1;

1:
  PastPrev:=Step;
  q_VA541:= TRUE;
  T_StepFW.IN:= TRUE;
  IF T_StepFW.Q THEN
     T_StepFW.IN := FALSE;
     Step:=2;
  END_IF;

2:
  PastPrev:=Step;
  q_VA401:= TRUE;
  T_StepFW.IN:= TRUE;
  IF T_StepFW.Q THEN
     T_StepFW.IN := FALSE;
     Step:=3;
  END_IF;

3:
  PastPrev:=Step;
  q_VA201:= TRUE;
  T_StepFW.IN:= TRUE;
  IF T_StepFW.Q THEN
     T_StepFW.IN := FALSE;
     Step:=4;
  END_IF;

4:
  PastPrev:=Step;
  q_VA301:= TRUE;
  T_StepFW.IN:= TRUE;
  IF T_StepFW.Q THEN
     T_StepFW.IN := FALSE;
     Step:=5;
  END_IF;

5:
  PastPrev:=Step;
  q_VA41:= TRUE;
  T_StepFW.IN:= TRUE;
  IF T_StepFW.Q THEN
     T_StepFW.IN := FALSE;
     Step:=6;
  END_IF;

6:
  PastPrev:=Step;
  q_VA11:= TRUE;
  T_StepFW.IN:= TRUE;
  IF T_StepFW.Q THEN
     T_StepFW.IN := FALSE;
     Step:=7;
  END_IF;

7:
  PastPrev:=Step;
  q_VA21:= TRUE;
  T_StepFW.IN:= TRUE;
  IF T_StepFW.Q THEN
     T_StepFW.IN := FALSE;
     Step:=8;
  END_IF;

8:
  PastPrev:=Step;
  q_VA31:= TRUE;
  T_StepFW.IN:= TRUE;
  IF T_StepFW.Q THEN
     T_StepFW.IN := FALSE;
     Step:=9;
  END_IF;

9:
  PastPrev:=Step;
  q_VA551:= TRUE;
  T_StepFW.IN:= TRUE;
  IF T_StepFW.Q THEN
     T_StepFW.IN := FALSE;
     Step:=10;
  END_IF;

10:
  PastPrev:=Step;
  q_VA501:= TRUE;
  T_StepFW.IN:= TRUE;
  IF T_StepFW.Q THEN
     T_StepFW.IN := FALSE;
     Step:=11;
  END_IF;

11:
  PastPrev:=Step;
  q_VA51:= TRUE;
  T_StepFW.IN:= TRUE;
  IF T_StepFW.Q THEN
     T_StepFW.IN := FALSE;
     Step:=12;
  END_IF;

12:
  PastPrev:=Step;
  q_VA511:= TRUE;
  T_StepFW.IN:= TRUE;
  IF T_StepFW.Q THEN
     T_StepFW.IN := FALSE;
     Step:=13;
  END_IF;

13:
  PastPrev:=Step;
  q_VA521:= TRUE;
  T_StepFW.IN:= TRUE;
  IF T_StepFW.Q THEN
     T_StepFW.IN := FALSE;
     Step:=14;
  END_IF;

14:
  PastPrev:=Step;
  q_VA531:= TRUE;
  T_StepFW.IN:= TRUE;
  IF T_StepFW.Q THEN
     T_StepFW.IN := FALSE;
     Step:=15;
  END_IF;

15:; (*выполнено*)
q_VisuMode:=0;



(*-----------------авария----------------*)
30:
	q_Red  :=TRUE;
	q_Sirena:=TRUE;
    IF AlarmReset THEN
       Step:= PastPrev;
    END_IF;
   q_VisuMode:=11;

END_CASE;


T_StepFW(PT:=T#5s);
END_FUNCTION_BLOCK

(* POU SwillWater, ST *)
FUNCTION_BLOCK SwillWater
VAR_INPUT
	i_Diag: BOOL;
	i_Pause: BOOL;
	i_fresh: BOOL;    (*полоскание вовзратной водой -0 , чистой - 1*)
	i_Block_Q4_out  : BOOL; (*блокировка выпуска для полоскания из Q4  - мин уровень и ph*)
	i_Block_Q4_in   : BOOL; (*блокировка подачи в Q4 - макс уровень и ph*)
	i_Ready_Route: BOOL; (*сигнал о готовности выбранного маршрута, если 0 - запрет старта процесса или в паузу *)
	i_FS: BOOL;       (*датчик протока на возврате*)
	i_Current_VolumeFC11: REAL;  (*текуший объем расходомера подачи*)

	i_TimeDelay           : DINT ; (*время задержки вкл/выкл клапанов и насосов*)
	i_TimeProcess         : DINT ; (*время мойки, мин*)

	i_RouteType           : DINT ; (*тип маршрута 1 - емкостной,0 - замкнутый*)
	i_PumpCapacity        : DINT ; (*производительность подающего насоса *)
	i_TimeDelayRetPump    : DINT ; (*время задержки включения насоса возврата*)
	i_TimeDelayRetFlow    : DINT ; (*время появления протока на возврате*)
	i_TimeAlarmBackFlow   : DINT ; (*время задержки аварии отсутсвия обратного протока*)

    Step: INT;
END_VAR
VAR_OUTPUT
	q_VA541: BOOL;
	q_VA401: BOOL;
	q_VA201: BOOL;
	q_VA301: BOOL;
	q_VA41 : BOOL;
	q_VA11 : BOOL;
	q_VA21 : BOOL;
	q_VA31 : BOOL;
	q_VA551: BOOL;
	q_VA501: BOOL;
	q_VA51 : BOOL;
	q_VA511: BOOL;
	q_VA521: BOOL;
	q_VA531: BOOL;
	q_P1   : BOOL;
	q_Red  : BOOL;
	q_Yellow : BOOL;
	q_Green  : BOOL;
	q_Sirena : BOOL;
	q_BackPump: BOOL;
	q_Heating_VR1: BOOL;
	q_AlarmBackFlow:BOOL;  (* авария протока на возврате*)
	q_Vis_tim_Process:BOOL;
	q_FC11_start: BOOL;	  (*старт подсчета импульсов*)
	q_ZeroCount_FC11: BOOL; (*обнуление счетчика*)
	q_SP_P1 : REAL;
	q_SP_VR1: REAL;
	q_VisuMode: INT;
END_VAR
(*
VAR RETAIN
	PastPrev       : INT;
	StepBackPump   : INT; (*задание режима работы возврата: 0 - отключено, 1 - возврата, 2 - пауза, 3 - докачка*)
	Step_Q4        : INT;   (*шаги переключения между Q1-Q4*)
	Last_Time_min  : DINT;  (*расчет оставшихся минут процесса*)
	Last_Time_sec  : DINT;  (*расчет оставшихся секунд процесса*)
END_VAR
*)
VAR

	PastPrev             AT %M*: INT;
	StepBackPump    AT %M*: INT; (*задание режима работы возврата: 0 - отключено, 1 - возврата, 2 - пауза, 3 - докачка*)
	Step_Q4              AT %M*: INT;   (*шаги переключения между Q1-Q4*)
	Last_Time_min     AT %M*: DINT;  (*расчет оставшихся минут процесса*)
	Last_Time_sec     AT %M*: DINT;  (*расчет оставшихся секунд процесса*)

	EndReturn            :BOOL;  (* окончание докачки из маршрута*)
	Return_OK            :BOOL;  (* таймера отсчитали, идет возврат - норма*)
	T_Delay   :TON;  (*служебный таймер*)
	T_BackPump:TON;  (*таймер задержки вклчения насоса возврата*)
	T_Process :TON;
	Return_Flow : BackPump; (*блок контроля и управления возвратом моющих средств*)

END_VAR
(*обнуление в начале скана*)
	q_VA541 := FALSE;  (*НО*)
	q_VA401 := FALSE;
	q_VA201 := FALSE;
	q_VA301 := FALSE;
	q_VA41  := FALSE;
	q_VA11  := FALSE;
	q_VA21  := FALSE;
	q_VA31  := FALSE;
	q_VA551 := FALSE;
	q_VA501 := FALSE;
	q_VA51  := FALSE;
	q_VA511 := FALSE;
	q_VA521 := FALSE;
	q_VA531 := FALSE;  (*НО*)
	q_P1 := FALSE;
    q_Green :=FALSE;
    q_Yellow :=FALSE;
    q_Red:=FALSE;
    q_Sirena :=FALSE;
	q_BackPump := FALSE;
    q_Heating_VR1 := FALSE;
    q_AlarmBackFlow := FALSE;
    q_Vis_tim_Process := FALSE;
	q_FC11_start := FALSE;
	q_ZeroCount_FC11 := FALSE;
	q_SP_P1 :=0.0 ;
	q_SP_VR1 :=0.0 ;

(*выход в аварию*)
IF i_Diag   THEN
   IF Step=0 THEN
      PastPrev:=0;
   END_IF;
   Step:=30;
END_IF;

(*выход в паузу*)
IF i_Pause   THEN
   IF Step=0 THEN
      PastPrev:=0;
   END_IF;
   Step:=35;
END_IF;

(*выход в паузу по неготовности маршрута*)
IF NOT i_Ready_Route THEN
   IF Step=0 THEN
      PastPrev:=0;
   END_IF;
   Step:=36;
END_IF;


CASE Step OF
0: (*обнуление*)
  T_Delay.IN:=FALSE;
  T_BackPump.IN:=FALSE;
  T_Process.IN:=FALSE;
  Step_Q4:=0;
  q_ZeroCount_FC11:=TRUE;

  StepBackPump:=0;
  Step:=1;

1: (*открытие клапанов, пуск насосов, подача в маршрут*)
  PastPrev:=Step;
  q_P1:=TRUE;
  q_SP_P1:=i_PumpCapacity;
  StepBackPump:=1;

      IF NOT i_fresh THEN  (*полоскание возвратной водой*)
        CASE Step_Q4 OF
        0: (*полоскание из Q4*)
           q_VA41:=TRUE;
           T_Delay.PT:=T#3s;
           T_Delay.IN:=i_Block_Q4_out;
           IF T_Delay.Q THEN
              Step_Q4:=1;
              T_Delay.IN:=FALSE;
           END_IF;
        1: (*переключение*)
           q_VA41:=TRUE;
           q_VA11:=TRUE;
           T_Delay.PT:=DINT_TO_TIME(i_TimeDelay*1000);
           T_Delay.IN:=TRUE;
           IF T_Delay.Q THEN
              Step_Q4:=2;
              T_Delay.IN:=FALSE;
           END_IF;
        2: (*полоскание из Q1, из Q4 заблокировано*)
           q_VA11:=TRUE;
           T_Delay.PT:=T#3s;
           T_Delay.IN:=NOT i_Block_Q4_out;
           IF T_Delay.Q THEN
              Step_Q4:=3;
              T_Delay.IN:=FALSE;
           END_IF;
        3: (*переключение*)
           q_VA41:=TRUE;
           q_VA11:=TRUE;
           T_Delay.PT:=DINT_TO_TIME(i_TimeDelay*1000);
           T_Delay.IN:=TRUE;
           IF T_Delay.Q THEN
              Step_Q4:=0;
              T_Delay.IN:=FALSE;
           END_IF;
         END_CASE;
      ELSE           (*полоскание чистой водой*)
         q_VA11 :=TRUE;
        CASE Step_Q4 OF
        0: (*возврат в Q4*)
           q_VA401:= TRUE;
           q_VA541:=TRUE; (*НО*)
           T_Delay.PT:=T#3s;
           T_Delay.IN:=i_Block_Q4_in;
           IF T_Delay.Q THEN
              Step_Q4:=1;
              T_Delay.IN:=FALSE;
           END_IF;
        1: (*переключение*)
           q_VA401:= TRUE;
           T_Delay.PT:=DINT_TO_TIME(i_TimeDelay*1000);
           T_Delay.IN:=TRUE;
           IF T_Delay.Q THEN
              Step_Q4:=2;
              T_Delay.IN:=FALSE;
           END_IF;
        2: (*возврат в канализацию, в Q4 заблокировано*)
           T_Delay.PT:=T#3s;
           T_Delay.IN:=NOT i_Block_Q4_in;
           IF T_Delay.Q THEN
              Step_Q4:=3;
              T_Delay.IN:=FALSE;
           END_IF;
        3: (*переключение*)
           q_VA401:= TRUE;
           T_Delay.PT:=DINT_TO_TIME(i_TimeDelay*1000);
           T_Delay.IN:=TRUE;
           IF T_Delay.Q THEN
              Step_Q4:=0;
              T_Delay.IN:=FALSE;
           END_IF;
        END_CASE;
      END_IF;


  IF Return_OK THEN (*возврта в норме*)
      T_Process.PT:=DINT_TO_TIME(i_TimeProcess*60000);
      Step:=2;
  END_IF;

  q_VisuMode:=2;

2: (*отсчет времени мойки*)
  PastPrev:=Step;
  q_P1:=TRUE;
  q_SP_P1:=i_PumpCapacity;
  StepBackPump:=1;

      IF NOT i_fresh THEN  (*полоскание возвратной водой*)
        CASE Step_Q4 OF
        0: (*полоскание из Q4*)
           q_VA41:=TRUE;
           T_Delay.PT:=T#3s;
           T_Delay.IN:=i_Block_Q4_out;
           IF T_Delay.Q THEN
              Step_Q4:=1;
              T_Delay.IN:=FALSE;
           END_IF;
        1: (*переключение*)
           q_VA41:=TRUE;
           q_VA11:=TRUE;
           T_Delay.PT:=DINT_TO_TIME(i_TimeDelay*1000);
           T_Delay.IN:=TRUE;
           IF T_Delay.Q THEN
              Step_Q4:=2;
              T_Delay.IN:=FALSE;
           END_IF;
        2: (*полоскание из Q1, из Q4 заблокировано*)
           q_VA11:=TRUE;
           T_Delay.PT:=T#3s;
           T_Delay.IN:=NOT i_Block_Q4_out;
           IF T_Delay.Q THEN
              Step_Q4:=3;
              T_Delay.IN:=FALSE;
           END_IF;
        3: (*переключение*)
           q_VA41:=TRUE;
           q_VA11:=TRUE;
           T_Delay.PT:=DINT_TO_TIME(i_TimeDelay*1000);
           T_Delay.IN:=TRUE;
           IF T_Delay.Q THEN
              Step_Q4:=0;
              T_Delay.IN:=FALSE;
           END_IF;
         END_CASE;
      ELSE           (*полоскание чистой водой*)
         q_VA11 :=TRUE;
        CASE Step_Q4 OF
        0: (*возврат в Q4*)
           q_VA401:= TRUE;
           q_VA541:=TRUE; (*НО*)
           T_Delay.PT:=T#3s;
           T_Delay.IN:=i_Block_Q4_in;
           IF T_Delay.Q THEN
              Step_Q4:=1;
              T_Delay.IN:=FALSE;
           END_IF;
        1: (*переключение*)
           q_VA401:= TRUE;
           T_Delay.PT:=DINT_TO_TIME(i_TimeDelay*1000);
           T_Delay.IN:=TRUE;
           IF T_Delay.Q THEN
              Step_Q4:=2;
              T_Delay.IN:=FALSE;
           END_IF;
        2: (*возврат в канализацию, в Q4 заблокировано*)
           T_Delay.PT:=T#3s;
           T_Delay.IN:=NOT i_Block_Q4_in;
           IF T_Delay.Q THEN
              Step_Q4:=3;
              T_Delay.IN:=FALSE;
           END_IF;
        3: (*переключение*)
           q_VA401:= TRUE;
           T_Delay.PT:=DINT_TO_TIME(i_TimeDelay*1000);
           T_Delay.IN:=TRUE;
           IF T_Delay.Q THEN
              Step_Q4:=0;
              T_Delay.IN:=FALSE;
           END_IF;
        END_CASE;
      END_IF;

     (*расчет времени для визуализ*)
    q_Vis_tim_Process := TRUE; (*визуализация полей времени*)
    Last_Time_min := (TIME_TO_DINT(T_Process.PT-T_Process.ET))/60000 ;
    Last_Time_sec := (TIME_TO_DINT(T_Process.PT-T_Process.ET)/1000) - Last_Time_min * 60 ;

   T_Process.in:=TRUE;
   IF T_Process.q THEN
      T_Process.in:=FALSE;
      Step:=3;
   END_IF;

  q_VisuMode:=3;

3: (*докачка из маршрута*)
  PastPrev:=Step;
  StepBackPump:=3;

(*задержка закрытия клапанов перед Р1*)
T_Process.in:=TRUE;
T_Process.PT:=T#5s;
IF NOT T_Process.q THEN
   q_VA11 :=i_fresh OR (NOT i_fresh AND i_Block_Q4_out);
   q_VA41 :=NOT i_fresh AND NOT i_Block_Q4_out;
END_IF;

      IF i_fresh THEN  (*полоскание чистой водой*)
        CASE Step_Q4 OF
        0: (*возврат в Q4*)
           q_VA401:= TRUE;
           q_VA541:=TRUE; (*НО*)
           T_Delay.PT:=T#3s;
           T_Delay.IN:=i_Block_Q4_in;
           IF T_Delay.Q THEN
              Step_Q4:=1;
              T_Delay.IN:=FALSE;
           END_IF;
        1: (*переключение*)
           q_VA401:= TRUE;
           T_Delay.PT:=DINT_TO_TIME(i_TimeDelay*1000);
           T_Delay.IN:=TRUE;
           IF T_Delay.Q THEN
              Step_Q4:=2;
              T_Delay.IN:=FALSE;
           END_IF;
        2: (*возврат в канализацию, в Q4 заблокировано*)
           T_Delay.PT:=T#3s;
           T_Delay.IN:=NOT i_Block_Q4_in;
           IF T_Delay.Q THEN
              Step_Q4:=3;
              T_Delay.IN:=FALSE;
           END_IF;
        3: (*переключение*)
           q_VA401:= TRUE;
           T_Delay.PT:=DINT_TO_TIME(i_TimeDelay*1000);
           T_Delay.IN:=TRUE;
           IF T_Delay.Q THEN
              Step_Q4:=0;
              T_Delay.IN:=FALSE;
           END_IF;
        END_CASE;
      END_IF;

     IF EndReturn THEN  (*закончилась откачка*)
         StepBackPump:=0;
         Step:=4;
     END_IF;

  q_VisuMode:=4;

4:; (*выполнено*)
     StepBackPump:=0;

(*-----------------авария----------------*)
30: (*авария*)
       q_VisuMode:=11;
       q_Red:=TRUE;
       q_Sirena :=TRUE;
       T_Process.IN := FALSE; (*остановка таймера процесса*)
       T_BackPump.IN:=FALSE;
       IF AlarmReset AND PastPrev=2  THEN
          T_Process.PT := DINT_TO_TIME(Last_Time_min*60000 + Last_Time_sec*1000);  (*уставка для таймера  в случае выхода в аварию*)
          Step := PastPrev;
       ELSIF AlarmReset AND PastPrev<>2 THEN
          Step := PastPrev;
       END_IF;

(*-----------------пауза----------------*)
35: (*пауза*)
       q_VisuMode:=12;
       q_Yellow:=TRUE;
       T_Process.IN := FALSE; (*остановка таймера процесса*)
       T_BackPump.IN:=FALSE;
       IF NOT i_Pause AND PastPrev=2  THEN
          T_Process.PT := DINT_TO_TIME(Last_Time_min*60000 + Last_Time_sec*1000);  (*уставка для таймера  в случае выхода в аварию*)
          Step := PastPrev;
       ELSIF NOT i_Pause AND PastPrev<>2 THEN
          Step := PastPrev;
       END_IF;

(*-----------------пауза - не готов маршрут----------------*)
36: (*пауза*)
       q_VisuMode:=18;
       q_Yellow:=TRUE;
       T_Process.IN := FALSE; (*остановка таймера процесса*)
       T_BackPump.IN:=FALSE;
       IF i_Ready_Route AND PastPrev=2  THEN
          T_Process.PT := DINT_TO_TIME(Last_Time_min*60000 + Last_Time_sec*1000);  (*уставка для таймера  в случае выхода в аварию*)
          Step := PastPrev;
       ELSIF i_Ready_Route AND PastPrev<>2 THEN
          Step := PastPrev;
       END_IF;

 END_CASE;

(*блок контроля и управления возвратом моющих средств*)
Return_Flow(
	i_AlarmPause:= (Step>=30),  (*в аварии или в паузе мойки или неготовности маршрута*)
	i_FS:= i_FS ,
	i_StepBackPump:= StepBackPump ,
	i_RouteType:= i_RouteType ,
	i_Current_VolumeFC11:= i_Current_VolumeFC11 ,
	i_TimeDelayRetPump:= i_TimeDelayRetPump ,
	i_TimeDelayRetFlow:= i_TimeDelayRetFlow ,
	i_TimeAlarmBackFlow:= i_TimeAlarmBackFlow ,
	q_BackPump=> q_BackPump ,
	q_AlarmBackFlow=> q_AlarmBackFlow ,
	q_EndReturn=>EndReturn  ,
      q_Return_OK=>Return_OK ,
	q_ZeroCount_FC11=> q_ZeroCount_FC11 ,
	q_FC11_start=> q_FC11_start );



T_Process();
T_BackPump();
T_Delay();
END_FUNCTION_BLOCK

(* POU BackPump, ST *)
FUNCTION_BLOCK BackPump (*блок контроля и управления возвратом моющих средств*)
VAR_INPUT
	i_AlarmPause			: BOOL;  (*остановка цикла по аварии или паузе Step=30, Step=35, Step=36*)
	i_FS					: BOOL;       (*датчик протока на возврате*)
	i_StepBackPump   		: INT; (*задание режима работы: 0 - отключено, 1 - старт возврата, 2 - пауза, 3 - докачка*)
	i_RouteType           		: DINT ; (*тип маршрута 1 - емкостной,0 - замкнутый*)
	i_Current_VolumeFC11	: REAL;  (*текуший объем расходомера подачи*)
	i_TimeDelayRetPump   	: DINT ; (*время задержки включения насоса возврата - объем подачи перед вкл*)
	i_TimeDelayRetFlow    	: DINT ; (*время появления протока на возврате*)
	i_TimeAlarmBackFlow   	: DINT ; (*время задержки аварии отсутсвия обратного протока*)
END_VAR

VAR_OUTPUT
	q_BackPump            	:BOOL;
	q_AlarmBackFlow     	:BOOL;  (* авария протока на возврате*)
	q_EndReturn            	:BOOL;  (* окончание докачки*)
	q_Return_OK            	:BOOL;  (* таймера отсчитали, идет возврат - норма*)
	q_ZeroCount_FC11   	:BOOL; (*обнуление расходомера*)
	q_FC11_start            	:BOOL;	(*старт подсчета импульсов*)
END_VAR

VAR
	Step  				AT %M* : INT;
	T_BackPump				:TON;  (*таймер задержки вклчения насоса возврата*)
END_VAR
(*обнуление в начале скана*)
q_BackPump := FALSE;
q_AlarmBackFlow := FALSE;
q_EndReturn := FALSE;
q_Return_OK := FALSE;
q_ZeroCount_FC11 := FALSE;
q_FC11_start := FALSE;

IF i_StepBackPump=0 THEN  (*выход из процесса*)
    Step := 0;
END_IF;


CASE i_RouteType OF

0: (*---------------------ЗАМКНУТЫЙ маршрут--------------*)
        IF NOT i_AlarmPause  THEN
            CASE  Step OF
            0: (*насос возврата и контроль выключены*)
                T_BackPump.IN:=FALSE;
                IF i_StepBackPump > 0 THEN  (*старт процесса*)
                    Step := 1;
                END_IF;
            1: (*переход*)
                Step := 2;
            2: (*контроль появления протока*)
                T_BackPump.PT:=DINT_TO_TIME(i_TimeDelayRetFlow*1000);
                T_BackPump.IN:=TRUE;
                IF T_BackPump.Q AND i_FS THEN  (*отсчитал таймер и сработал датчик*)
                    T_BackPump.IN:=FALSE;
                     Step:=3;
                ELSIF T_BackPump.Q AND NOT i_FS THEN (*в аварию*)
                      q_AlarmBackFlow:=TRUE;
                END_IF;
                IF i_StepBackPump=3 THEN  (*на докачку*)
                    T_BackPump.IN:=FALSE;
                    Step := 4;
                END_IF;
             3: (*контроль возврата в процессе мойки*)
                q_Return_OK:=TRUE;
                T_BackPump.PT:=DINT_TO_TIME(i_TimeAlarmBackFlow*1000);
                T_BackPump.IN:=NOT i_FS;
                IF T_BackPump.Q  THEN (*в аварию*)
                    q_AlarmBackFlow:=TRUE;
                END_IF;
                IF i_StepBackPump=3 THEN (*на докачку*)
                   T_BackPump.IN:=FALSE;
                   Step :=4;
                END_IF;
             4: (*докачка*)
                T_BackPump.PT:=DINT_TO_TIME(i_TimeAlarmBackFlow*1000);
                T_BackPump.IN:=NOT i_FS;
                IF T_BackPump.Q  THEN
                    q_EndReturn := TRUE;
                END_IF;
            END_CASE;
         ELSE (*авария или пауза*)
             T_BackPump.IN:=FALSE;
             IF ((Step > 1) AND (Step < 4)) THEN (*в случае аварии во время процесса отсчет задержки появл протока как при старте*)
                 Step := 2;
             END_IF;
          END_IF;

1: (*---------------------ЕМКОСТНОЙ маршрут--------------*)
        IF NOT i_AlarmPause  THEN
            CASE  Step OF
            0: (*насос возврата и контроль выключены*)
                T_BackPump.IN:=FALSE;
                IF i_StepBackPump > 0 THEN  (*старт процесса*)
                    q_ZeroCount_FC11:=TRUE; (*обнулили счетчик*)
                    Step := 1;
                END_IF;
             1: (*отсчет задержки включения насоса НВ*)
                 q_FC11_start:=TRUE; (*контроль по объему*)
                 IF (i_Current_VolumeFC11>=i_TimeDelayRetPump) THEN (*отсчитали объем*)
                     T_BackPump.IN:=FALSE;
                     q_ZeroCount_FC11:=TRUE; (*обнулили счетчик*)
                     Step:=2;
                  END_IF;
            2: (*включение НВ. контроль появления протока*)
                q_BackPump:= (i_StepBackPump=1);  (*НВ работает если не пауза*)
                T_BackPump.PT:=DINT_TO_TIME(i_TimeDelayRetFlow*1000);
                T_BackPump.IN:= (i_StepBackPump=1);  (*контроль возврата если не пауза*);
                IF T_BackPump.Q AND i_FS THEN  (*отсчитал таймер и сработал датчик*)
                    T_BackPump.IN:=FALSE;
                      Step:=3;
                ELSIF T_BackPump.Q AND NOT i_FS THEN (*в аварию*)
                      q_AlarmBackFlow:=TRUE;
                END_IF;
                IF i_StepBackPump=3 THEN  (*на докачку*)
                    T_BackPump.IN:=FALSE;
                    Step := 4;
                END_IF;
             3: (*контроль возврата в процессе мойки*)
                q_Return_OK:=TRUE;
                q_BackPump:= TRUE;
                T_BackPump.PT:=DINT_TO_TIME(i_TimeAlarmBackFlow*1000);
                T_BackPump.IN:=NOT i_FS;
                IF T_BackPump.Q  THEN (*в аварию*)
                    q_AlarmBackFlow:=TRUE;
                END_IF;
                IF i_StepBackPump=2 THEN  (*пауза*)
                   T_BackPump.IN:=FALSE;
                   Step :=2;
                ELSIF i_StepBackPump=3 THEN (*на докачку*)
                   T_BackPump.IN:=FALSE;
                   Step :=4;
                END_IF;
             4: (*докачка*)
                q_BackPump:= TRUE;
                T_BackPump.PT:=DINT_TO_TIME(i_TimeAlarmBackFlow*1000);
                T_BackPump.IN:=NOT i_FS;
                IF T_BackPump.Q  THEN
                    q_EndReturn := TRUE;
                END_IF;
            END_CASE;
         ELSE (*авария или пауза*)
             T_BackPump.IN:=FALSE;
             IF ((Step > 1) AND (Step < 4)) THEN (*в случае аварии во время процесса отсчет задержки появл протока как при старте*)
                 Step := 2;
             END_IF;
         END_IF;



END_CASE;


T_BackPump();
END_FUNCTION_BLOCK

(* POU WashSolution, ST *)
FUNCTION_BLOCK WashSolution  (*мойка рвстворами*)
VAR_INPUT
	i_Diag: BOOL;
	i_Diag_Preparation: BOOL;
	i_Pause: BOOL;
	i_Block_Q4_out  : BOOL; (*блокировка выпуска для полоскания из Q4  - мин уровень и ph*)
	i_Block_Q4_in   : BOOL; (*блокировка подачи в Q4 - макс уровень и ph*)
	i_Block_SolPrep : BOOL; (*блокировка подготовки раствора - идет мойка этим же р-ром по другому контуру*)
	i_Alarm_LSmin: BOOL;   (*авария нижнего уровня в баке концентрата*)
	i_Ready_Route: BOOL; (*сигнал о готовности выбранного маршрута, если 0 - запрет старта процесса или в паузу *)
	i_Alk: BOOL;       (*мойка щелочью*)

	i_FS: BOOL;       (*датчик протока на возврате*)
	i_LSL: BOOL;      (*датчик уровня в циркуляционном баке*)
	i_LSM: BOOL;      (*датчик уровня в циркуляционном баке*)
	i_LSH: BOOL;      (*датчик уровня в циркуляционном баке*)
	i_Mixing: BOOL;   (*перемешивание перед мойкой*)

	i_TE1: REAL;      (*температура на подаче*)
	i_TE2: REAL;      (*температура на возврате*)
	i_TE_tank: REAL;  (*температура в танке раствора*)
	i_LE_tank: REAL;  (*уровень в танке раствора*)
	i_QE : REAL;      (*расчитанная концентрация % раствора*)
	i_QE_priv : REAL; (*приведенная проводимость к температуре*)
	i_Current_VolumeFC11: REAL;  (*текуший объем расходомера подачи*)

	i_MaxCondPrep: REAL;  (*максимальная проводимость раствора при подготовке*)
	i_MinCondPrep: REAL;  (*минимальная проводимость раствора при подготовке*)
	i_MaxTempPrep: REAL;  (*максимальная темп при подготовке*)
	i_MinTempPrep: REAL;  (*минимальная темп при подготовке*)
	i_LvlPrep: INT;       (*заданный уровень в баке раствора при подготовке*)
	Cond_Q4: REAL;        (*концентрация для перехода с/на бак Q4*)

	i_TimeDelay           : DINT ; (*время задержки вкл/выкл клапанов и насосов*)
	i_Time_LSH_on         : DINT ; (*время задержки срабатывания датчика верх уровня цирк бака*)
	i_Time_LSM_on         : DINT ; (*время задержки срабатывания датчика сред уровня цирк бака*)
	i_Time_LSM_off        : DINT ; (*время задержки отключения датчика сред уровня цирк бака*)
	i_Time_LSL_off        : DINT ; (*время задержки отключения датчика ниж уровня цирк бака*)
	i_TimeProcess         : DINT ; (*время мойки*)
	i_TempProcess         : REAL ; (*температура мойки*)

	i_RouteType           : DINT ; (*тип маршрута 1 - емкостной,0 - замкнутый*)
	i_PumpCapacity        : DINT ; (*производительность подающего насоса *)
	i_TimeDelayRetPump    : DINT ; (*время задержки включения насоса возврата - объем подачи перед вкл*)
	i_TimeDelayRetFlow    : DINT ; (*время появления протока на возврате*)
	i_TimeAlarmBackFlow   : DINT ; (*время задержки аварии отсутсвия обратного протока*)
	i_Using_Q5          :DINT;       (*использование циркуляционного бака на мойках растворами и водой, 1 - использовать*)

    Step: INT;
END_VAR
VAR_OUTPUT
	q_VA541: BOOL;
	q_VA401: BOOL;
	q_VA201: BOOL;
	q_VA41 : BOOL;
	q_VA11 : BOOL;
	q_VA21 : BOOL;
	q_VA551: BOOL;
	q_VA501: BOOL;
	q_VA51 : BOOL;
	q_VA511: BOOL;
	q_VA521: BOOL;
	q_VA531: BOOL;
	q_VE11 : BOOL;
	q_P1   : BOOL;
	q_P10  : BOOL;
	q_Red  : BOOL;
	q_Yellow : BOOL;
	q_Green  : BOOL;
	q_Sirena : BOOL;
	q_BackPump: BOOL;
	q_Heating_VR1: BOOL;
	q_AlarmBackFlow:BOOL;  (* авария протока на возврате*)
	q_AlarmQ4: BOOL;       (*неготовность танка Q4, пауза процесса*)
	q_Alarm_Empty_Q5: BOOL;(*авария опустошения цирк бака при работе на замкн маршруте*)
	q_Vis_tim_Process:BOOL;
	q_FC11_start: BOOL;	  (*старт подсчета импульсов*)
	q_ZeroCount_FC11: BOOL; (*обнуление счетчика*)
	q_Block_Solution : BOOL; (*блокировка использования раствора другими контурами*)
	q_SP_P1 : REAL;
	q_SP_VR1: REAL;
	q_VisuMode: INT;
END_VAR

VAR

	PastPrev              AT %M*: INT;
	StepBackPump    AT %M*: INT; (*задание режима работы возврата: 0 - отключено, 1 - старт возврата, 2 - пауза, 3 - докачка*)
	Last_Time_min     AT %M*: DINT;  (*расчет оставшихся минут процесса*)
	Last_Time_sec     AT %M* : DINT;  (*расчет оставшихся секунд процесса*)

	EndReturn            :BOOL;  (* окончание докачки из маршрута*)
	Return_OK            :BOOL;  (* таймера отсчитали, идет возврат - норма*)
      Start_Control_Q4   :BOOL ;   (*старт процесса контроля потока в танк возвратной воды Q4 *)
	ModeControl_Q5   : INT;    (*режим поддержания уровня в цирк баке: 0 - выкл, 1 - во время мойки через цирк бак, 2 - при промывке и вытесн через цирк бак*)
	Step_Q5: INT;  (*шаги контроля уровня в цирк баке*)
	T_Delay   :TON;  (*служебный таймер*)
	T_LSL_off :TON;
	T_LSH_on  :TON;
	T_LSM_on  :TON;
	T_LSM_off :TON;
	T_Process :TON;
	Preparation:SolutionPrepar;
	Return_Flow : BackPump; (*блок контроля и управления возвратом моющих средств*)
	Control_Q4 :Q4_Level;   (*блок контроля потока в танк возвратной воды Q4*)
	Control_Q5 :Q5_Level;  (*блок поддержания уровня в циркуляционном баке во время мойки и при откачке*)
END_VAR
(*обнуление в начале скана*)
	q_VA541 := FALSE;  (*НО*)
	q_VA401 := FALSE;
	q_VA201 := FALSE;
	q_VA41  := FALSE;
	q_VA11  := FALSE;
	q_VA21  := FALSE;
	q_VA551 := FALSE;
	q_VA501 := FALSE;
	q_VA51  := FALSE;
	q_VA511 := FALSE;
	q_VA521 := FALSE;
	q_VA531 := FALSE;  (*НО*)
	q_VE11  := FALSE;
	q_P1 := FALSE;
	q_P10 := FALSE;
      q_Green :=FALSE;
      q_Yellow :=FALSE;
      q_Red:=FALSE;
      q_Sirena :=FALSE;
	q_BackPump := FALSE;
      q_Heating_VR1 := FALSE;
      q_AlarmBackFlow := FALSE;
      q_AlarmQ4:=FALSE;
      q_Alarm_Empty_Q5:=FALSE;
      q_Vis_tim_Process := FALSE;
	q_FC11_start := FALSE;
	q_ZeroCount_FC11 := FALSE;
      q_Block_Solution:=FALSE;
      Start_Control_Q4 := FALSE;
	q_SP_P1 :=0.0 ;
	q_SP_VR1 :=0.0 ;
      ModeControl_Q5 := 0;


(*выход в аварию*)
IF i_Diag   THEN
   IF Step=0 THEN
      PastPrev:=0;
   END_IF;
   Step:=30;
END_IF;

(*выход в паузу*)
IF i_Pause   THEN
   IF Step=0 THEN
      PastPrev:=0;
   END_IF;
   Step:=35;
END_IF;

(*выход в паузу по неготовности маршрута*)
IF NOT i_Ready_Route THEN
   IF Step=0 THEN
      PastPrev:=0;
   END_IF;
   Step:=36;
END_IF;

CASE Step OF
0: (*обнуление*)
  T_Delay.IN:=FALSE;
  T_Process.IN:=FALSE;
  q_ZeroCount_FC11:=TRUE;
  StepBackPump := 0;
  IF i_Mixing AND NOT i_Block_SolPrep THEN (*если мешаем и нет мойки этим же р-ром по др контурам*)
      IF i_LE_tank < i_LvlPrep THEN  (*уровень в танке р-ра менее заданного - сразу на подготовку*)
           Preparation.Step:=0;
           Step:=3;
      ELSE                                       (*уровень в норме - на перемешивание и проверку концентрации*)
           Step:=1;
      END_IF;
  ELSE                                  (*подача в маршрут*)
     Step:=5 ;
  END_IF;


1: (*перемешивание,проверка раствора*)
  PastPrev:=Step;
  q_VA21:=TRUE;
  q_VA521:=TRUE;
  q_VA531:=TRUE; (*НО*)
  q_VA541:=TRUE; (*НО*)
  q_VA201:=TRUE;
  q_P1:=TRUE;
  q_SP_P1:=FlowPrep;
  q_Block_Solution:=TRUE;  (*блокировка использования раствора другими контурами*)
  StepBackPump := 0; (*выключить вовзрат и контроль возврата*)

     (*расчет времени для визуализ*)
    q_Vis_tim_Process := TRUE; (*визуализация полей времени*)
    Last_Time_min := (TIME_TO_DINT(T_Process.PT-T_Process.ET))/60000 ;
    Last_Time_sec := (TIME_TO_DINT(T_Process.PT-T_Process.ET)/1000) - Last_Time_min * 60 ;

   T_Process.PT:=DINT_TO_TIME(TimeMixPrep*1000);
   T_Process.in:=TRUE;
   IF T_Process.q AND i_QE<i_MinCondPrep THEN  (*если концентрация ниже минимальной то сразу на шаг набора концентрации*)
      T_Process.in:=FALSE;
      Preparation.Step:=5;
      Step:=3;
   ELSIF T_Process.q AND i_QE>=i_MinCondPrep THEN  (*концентарция в норме*)
      T_Process.in:=FALSE;
      Step:=4 ;
   END_IF;

  q_VisuMode:=6;

2: (*остановка перед подготовкой - перескакиваем*)
  PastPrev:=Step;
  q_VA21:=TRUE;
  q_VA521:=TRUE;
  q_VA531:=TRUE; (*НО*)
  q_VA541:=TRUE; (*НО*)
  q_VA201:=TRUE;
  q_Block_Solution:=TRUE;  (*блокировка использования раствора другими контурами*)
  StepBackPump := 0; (*выключить вовзрат и контроль возврата*)

  T_Delay.PT:=DINT_TO_TIME(i_TimeDelay*1000);
  T_Delay.IN:=TRUE;
  IF T_Delay.Q THEN
     T_Delay.IN:=FALSE;
     Step:=3;
  END_IF;

  q_VisuMode:=6;

3: (*подготовка растворов*)
  PastPrev:=Step;
  q_Block_Solution:=TRUE;  (*блокировка использования раствора другими контурами*)
  StepBackPump := 0; (*выключить возврат и контроль возврата*)

  Preparation.i_Diag:=i_Diag_Preparation;
Preparation(
	i_Pause:=i_Pause ,
	i_Block_Q4_out:=i_Block_Q4_out,
	i_Block_Q4_in:=i_Block_Q4_in ,
	i_Alarm_LSmin:=i_Alarm_LSmin ,
	i_Alk:=i_Alk,
	i_FS:=i_FS ,
	i_TE1:=i_TE1 ,
	i_TE2:=i_TE2 ,
	i_TE_tank:=i_TE_tank ,
	i_LE_tank:=i_LE_tank ,
	i_QE:=i_QE ,
	i_QE_priv:=i_QE_priv ,
	i_TimeDelay:=i_TimeDelay ,
	i_MaxCondPrep:=i_MaxCondPrep ,
	i_MinCondPrep:=i_MinCondPrep ,
	i_MaxTempPrep:=i_MaxTempPrep ,
	i_MinTempPrep:=i_MinTempPrep ,
	i_LvlPrep:=i_LvlPrep ,
	q_VA541=>q_VA541 ,
	q_VA401=>q_VA401 ,
	q_VA201=>q_VA201 ,
	q_VA41=>q_VA41 ,
	q_VA11=>q_VA11 ,
	q_VA21=>q_VA21 ,
	q_VA551=>q_VA551 ,
	q_VA501=>q_VA501 ,
	q_VA51=>q_VA51 ,
	q_VA511=>q_VA511 ,
	q_VA521=>q_VA521 ,
	q_VA531=>q_VA531 ,
	q_VE11=>q_VE11 ,
	q_P1=>q_P1 ,
	q_P10=>q_P10 ,
	q_Red=>q_Red ,
	q_Yellow=>q_Yellow ,
	q_Green=>q_Green ,
	q_Sirena=>q_Sirena ,
	q_Heating_VR1=>q_Heating_VR1 ,
	q_AlarmBackFlow=>q_AlarmBackFlow ,
	q_Vis_tim_Process=>q_Vis_tim_Process ,
	q_SP_P1=>q_SP_P1 ,
	q_SP_VR1=>q_SP_VR1 ,
	q_VisuMode=>q_VisuMode );
    Last_Time_min := Preparation.Last_Time_min;
    Last_Time_sec := Preparation.Last_Time_sec;

    IF Preparation.Step=6 AND i_TE_tank>=(i_MaxTempPrep-1) THEN
       T_Delay.IN:=FALSE;
       Step:=4;
    END_IF;

4: (*переключение в маршрут*)
  PastPrev:=Step;
  q_VA21:=TRUE;
  q_VA521:=TRUE;
  q_VA541:=TRUE; (*НО*)
  q_VA201:=TRUE;
  q_VA401:=TRUE;
  q_P1:=TRUE;
  q_SP_P1:=FlowPrep;
  StepBackPump := 0; (*выключить возврат и контроль возврата*)

  T_Delay.PT:=DINT_TO_TIME(i_TimeDelay*1000);
  T_Delay.IN:=TRUE;
  IF T_Delay.Q THEN
     T_Delay.IN:=FALSE;
     Step:=5;
  END_IF;

  q_VisuMode:=2;

5: (*подача в маршрут*)
  PastPrev:=Step;
  q_VA21:=TRUE;
  q_VA541:=TRUE; (*НО*)
  q_VA401:=TRUE;
  q_VA511:=(i_Using_Q5=1);
  q_P1:=TRUE;
  q_SP_P1:=i_PumpCapacity;
  StepBackPump:=1; (*включен возврат и контроль возврата*)

  IF Return_OK THEN (*возврат в норме. за контрольное время протока остатки р-ра в трубах CIP-мойки уйдут в бак Q4 *)
     Step:=6;
  END_IF;

  q_VisuMode:=2;


6: (*ожидание концентрации*)
  PastPrev:=Step;
  q_VA21:=TRUE;
  q_VA541:=TRUE; (*НО*)
  q_VA401:=TRUE;
  q_VA511:=(i_Using_Q5=1);
  q_P1:=TRUE;
  q_SP_P1:=i_PumpCapacity;
  q_Heating_VR1:=q_P1;
  q_SP_VR1 := i_TempProcess;
  StepBackPump:=1; (*включен возврат и контроль возврата*)

  T_Delay.PT:=T#2s;
  T_Delay.IN:=i_QE>Cond_Q4; (*достигнута концентрация перехода с бака Q4*)
  IF T_Delay.Q THEN
     T_Delay.IN:=FALSE;
     Step:=7;
  END_IF;

  q_VisuMode:=9;


7: (*переключение на цирк бак / или на танк раствора*)
  PastPrev:=Step;
  q_VA21:=TRUE;
  q_VA541:=TRUE; (*НО*)
  q_VA501:=(i_Using_Q5=1); (*мойка через цирк бак*)
  q_VA201:=(i_Using_Q5=0); (*мойка через танк раствора*)
  q_VA401:=TRUE;
  q_P1:=TRUE;
  q_SP_P1:=i_PumpCapacity;
  q_Heating_VR1:=TRUE;
  q_SP_VR1 := i_TempProcess;
  StepBackPump:=1; (*включен возврат и контроль возврата*)

  T_Delay.PT:=DINT_TO_TIME(i_TimeDelay*1000);
  T_Delay.IN:=TRUE;
  IF T_Delay.Q THEN
     T_Delay.IN:=FALSE;
     IF (i_Using_Q5=1) THEN  (*мойка через цирк бак*)
         Step:=8;
     ELSE
         Step := 10 ; (*если через танк то на догрев*)
     END_IF;
  END_IF;

  q_VisuMode:=9;

8: (*заполнение цирк бака*)
  PastPrev:=Step;
  q_VA21:=TRUE;
  q_VA541:=TRUE; (*НО*)
  q_VA501:=TRUE;
  q_P1:=TRUE;
  q_SP_P1:=i_PumpCapacity;
  q_Heating_VR1:=TRUE;
  q_SP_VR1 := i_TempProcess;
  StepBackPump:=1; (*включен возврат и контроль возврата*)

  IF T_LSM_on.Q THEN
     Step:=9;
  END_IF;

  q_VisuMode:=10;

9: (*переключение*)
  PastPrev:=Step;
  q_VA21:=TRUE;
  q_VA51:=TRUE;
  q_VA541:=TRUE; (*НО*)
  q_VA501:=TRUE;
  q_P1:=TRUE;
  q_SP_P1:=i_PumpCapacity;
  q_Heating_VR1:=TRUE;
  q_SP_VR1 := i_TempProcess;
  StepBackPump:=1; (*включен возврат и контроль возврата*)

  T_Delay.PT:=DINT_TO_TIME(i_TimeDelay*1000);
  T_Delay.IN:=TRUE;
  IF T_Delay.Q THEN
     T_Delay.IN:=FALSE;
     Step:=10;
  END_IF;

  q_VisuMode:=10;

10: (*догрев*)
  PastPrev:=Step;
  q_VA541:=TRUE; (*НО*)
  q_SP_P1:=i_PumpCapacity;
  q_Heating_VR1:=TRUE;
  q_SP_VR1 := i_TempProcess;

  IF (i_Using_Q5=1) THEN  (*мойка через цирк бак*)
      q_VA501:=TRUE;
      ModeControl_Q5 := 1; (*поддержание уровня в цирк баке во время мойки через цирк бак, контроль насоса Р1 и VA51*)

  ELSE         (*мойка через танк раствора*)
         q_VA21:=TRUE;
         q_VA201:=TRUE;
         q_P1:=TRUE;
         StepBackPump:=1; (*включен возврат и контроль возврата*)
 END_IF;

   IF i_TE1>(i_TempProcess-2.0) THEN  (*достигли заданную температуру*)
      T_Process.PT:=DINT_TO_TIME(i_TimeProcess*60000);
      Step:=11;
   END_IF;

  q_VisuMode:=8;

11: (*отсчет времени мойки*)
  PastPrev:=Step;
  q_VA541:=TRUE; (*НО*)
  q_SP_P1:=i_PumpCapacity;
  q_Heating_VR1:=TRUE;
  q_SP_VR1 := i_TempProcess;

  IF (i_Using_Q5=1) THEN  (*мойка через цирк бак*)
      q_VA501:=TRUE;
      ModeControl_Q5 := 1; (*поддержание уровня в цирк баке во время мойки через цирк бак, контроль насоса Р1 и q_VA51*)

  ELSE         (*мойка через танк раствора*)
         q_VA21:=TRUE;
         q_VA201:=TRUE;
         q_P1:=TRUE;
         StepBackPump:=1; (*включен возврат и контроль возврата*)
 END_IF;

     (*расчет времени для визуализ*)
    q_Vis_tim_Process := TRUE; (*визуализация полей времени*)
    Last_Time_min := (TIME_TO_DINT(T_Process.PT-T_Process.ET))/60000 ;
    Last_Time_sec := (TIME_TO_DINT(T_Process.PT-T_Process.ET)/1000) - Last_Time_min * 60 ;

   T_Process.in:=TRUE;
   IF T_Process.Q  THEN
       T_Process.in:=FALSE;
       IF i_Using_Q5 = 1 THEN (*если мылись через цирк бак*)
          Step:=12;
       ELSE                (*если мылись через танк раствора*)
          Step:=14;
       END_IF;
   END_IF;

  q_VisuMode:=3;

12: (*переключение. после мойки через цирк бак*)
  PastPrev:=Step;
  q_VA51:=TRUE;
  q_VA541:=TRUE; (*НО*)
  q_VA501:=TRUE;
  q_VA201:=TRUE;
  q_P1:=TRUE;
  q_SP_P1:=i_PumpCapacity;
  StepBackPump:=1; (*включен возврат и контроль возврата*)

  T_Delay.PT:=DINT_TO_TIME(i_TimeDelay*1000);
  T_Delay.IN:=TRUE;
  IF T_Delay.Q THEN
     T_Delay.IN:=FALSE;
     Step:=13;
  END_IF;

  q_VisuMode:=4;

13: (*откачка из цирк бака. после мойки через цирк бак*)
  PastPrev:=Step;
  q_VA51:=TRUE;
  q_VA541:=TRUE; (*НО*)
  q_VA201:=TRUE;
  q_P1:=TRUE;
  q_SP_P1:=i_PumpCapacity;
  StepBackPump:=1; (*включен возврат и контроль возврата*)

  IF T_LSL_off.Q AND NOT i_LSM THEN
      StepBackPump:=3;
      Step:=14;
  END_IF;

  q_VisuMode:=4;

14: (*откачка из маршрута*)
  PastPrev:=Step;
  q_VA541:=TRUE; (*НО*)
  q_VA201:=TRUE;
  StepBackPump:=3; (*откачка из маршрута*)

  T_Delay.PT:=DINT_TO_TIME(i_TimeDelay*1000); (*таймер задержки закрытия клапанов*)
  T_Delay.IN:=TRUE;

  IF i_Using_Q5=1 THEN (*мылись через цирк бак*)
        q_VA51:=NOT T_Delay.Q;  (*задержка закрытия клапана*)
        q_VA511:=TRUE;  (*сливаем остатки из цирк бака*)
  ELSE
        q_VA21 := NOT T_Delay.Q ;  (*задержка закрытия клапана*)
  END_IF;

      IF EndReturn  THEN (*докачали из маршрута*)
          T_Delay.IN:= FALSE;
         StepBackPump:=0; (*выключить вовзрат и контроль возврата*)
         Step:=15;
      END_IF;

  q_VisuMode:=13;


15: (*вытеснение раствора в бак раствора*)
  PastPrev:=Step;
  q_VA541:=TRUE; (*НО*)
  q_VA201:=TRUE;
  q_P1:=TRUE;
  q_SP_P1:=i_PumpCapacity;
  StepBackPump:=1; (*включен возврат и контроль возврата*)

  IF i_Using_Q5=1 THEN       (*мылись через цирк бак*)
      ModeControl_Q5 := 2; (*поддержание уровня в цирк баке при промывке и вытесн через цирк бак*)
  ELSE                 (*мылись через танк раствора, вода из танка Q1*)
       q_VA11:=TRUE;
  END_IF;


  IF i_QE<Cond_Q4 THEN  (*снизилась концентрация*)
     Step:=16;
  END_IF;

  q_VisuMode:=13;

16: (*вытеснение раствора в бак Q4*)
  PastPrev:=Step;
  q_VA541:=TRUE; (*НО*)
  q_VA401:=TRUE;
  q_P1:=TRUE;
  q_SP_P1:=i_PumpCapacity;
  StepBackPump:=1; (*включен возврат и контроль возврата*)

  T_Delay.PT:=DINT_TO_TIME(i_TimeDelay*1000);
  T_Delay.IN:=TRUE;
  q_VA201:=NOT T_Delay.Q; (*задержка закрытия клапана*)

    IF i_Using_Q5=1 THEN       (*мылись через цирк бак*)
        ModeControl_Q5 := 2; (*поддержание уровня в цирк баке при промывке и вытесн через цирк бак*)
   ELSE           (*мылись через танк раствора, вода из танка Q1*)
        q_VA11 :=TRUE;
   END_IF;

  IF i_QE_priv<5.0 THEN  (*концентрация снизилась до уровня воды*)
      T_Delay.IN:=FALSE;
      IF (i_Using_Q5=1) AND Control_Q5.Step_Q5<>1 AND Control_Q5.Step_Q5<>4 THEN (*если нет переключения клапанов цирк бака*)
           Step_Q5 := Control_Q5.Step_Q5 ; (*присваиваем номер шага*)
           Step:=17;
      ELSIF  (i_Using_Q5<>1) THEN
           Step := 18;
      END_IF;
  END_IF;

  q_VisuMode:=13;


17: (*опустошение цирк бака - мойка через цирк бак*)
  PastPrev:=Step;
  q_VA541:=TRUE; (*НО*)
  q_VA401:=TRUE;
  q_P1:=TRUE;
  q_SP_P1:=i_PumpCapacity;
  StepBackPump:=1; (*включен возврат и контроль возврата*)

      (*поддержание уровня в цирк баке*)
      CASE Step_Q5 OF
      0: (*заполнение цирк бака*)
         q_VA11 :=TRUE;
         Step_Q5:=1;
      1: (*переключение*)
         q_VA51:=TRUE;
         q_VA11:=TRUE;
         T_Delay.PT:=DINT_TO_TIME(i_TimeDelay*1000);
         T_Delay.IN:=TRUE;
         IF T_Delay.Q THEN
            T_Delay.IN:=FALSE;
            Step_Q5:=2;
         END_IF;
      2: (*на среднем*)
         q_VA51:=TRUE;
         IF T_LSH_on.Q THEN
            Step_Q5:=3;
         ELSIF T_LSL_off.Q AND NOT i_LSM THEN
            Step_Q5:=4;
         END_IF;
      3: (*на верхнем*)
         q_VA51:=TRUE;
         IF T_LSM_off.Q THEN
            Step_Q5:=2;
         END_IF;
      4: (*переключение*)
         q_VA51:=TRUE;
         T_Delay.IN:=FALSE;
         Step:=18;
      END_CASE;


  q_VisuMode:=4;

18: (*докачка из маршрута*)
  PastPrev:=Step;
  q_VA541:=TRUE; (*НО*)
  q_VA401:=TRUE;
  StepBackPump:=3; (*откачка из маршрута*)

(*задержка закрытия клапанов перед Р1*)
  T_Delay.PT:=T#5s;
  T_Delay.IN:=TRUE;
  q_VA51:=NOT T_Delay.Q AND (i_Using_Q5=1); (*была мойка через цирк бак*)
  q_VA11:=NOT T_Delay.Q AND (i_Using_Q5<>1); (*была мойка через танк раствора*)


      IF EndReturn THEN
          T_Delay.IN:= FALSE;
         StepBackPump := 0; (*выключить вовзрат и контроль возврата*)
         Step:=19;
      END_IF;

  q_VisuMode:=4;

19: (*выполнено*)
  q_VisuMode:=1;
 StepBackPump := 0; (*выключить вовзрат и контроль возврата*)



(*-----------------авария----------------*)
30: (*авария*)
       q_VisuMode:=11;
       q_Red:=TRUE;
       q_Sirena :=TRUE;
       T_Process.IN := FALSE; (*остановка таймера процесса*)
       IF AlarmReset AND PastPrev=11  THEN
          T_Process.PT := DINT_TO_TIME(Last_Time_min*60000 + Last_Time_sec*1000);  (*уставка для таймера  в случае выхода в аварию*)
          Step := PastPrev;
       ELSIF AlarmReset AND PastPrev<>11 THEN
          Step := PastPrev;
       END_IF;

(*-----------------пауза----------------*)
35: (*пауза*)
       q_VisuMode:=12;
       q_Yellow:=TRUE;
       T_Process.IN := FALSE; (*остановка таймера процесса*)
       IF NOT i_Pause AND PastPrev=11  THEN
          T_Process.PT := DINT_TO_TIME(Last_Time_min*60000 + Last_Time_sec*1000);  (*уставка для таймера  в случае выхода в аварию*)
          Step := PastPrev;
       ELSIF NOT i_Pause AND PastPrev<>11 THEN
          Step := PastPrev;
       END_IF;

(*-----------------пауза - не готов маршрут----------------*)
36: (*пауза*)
       q_VisuMode:=18;
       q_Yellow:=TRUE;
       T_Process.IN := FALSE; (*остановка таймера процесса*)
       IF i_Ready_Route AND PastPrev=11  THEN
          T_Process.PT := DINT_TO_TIME(Last_Time_min*60000 + Last_Time_sec*1000);  (*уставка для таймера  в случае выхода в аварию*)
          Step := PastPrev;
       ELSIF i_Ready_Route AND PastPrev<>11 THEN
          Step := PastPrev;
       END_IF;

 END_CASE;

(*блок поддержания уровня в циркуляционном баке во время мойки и при откачке*)
Control_Q5(
	i_P1:= q_P1,
	i_VA551:= q_VA551 ,
	i_VA11:= q_VA11 ,
	i_VA51:= q_VA51 ,
	i_LSL:= i_LSL ,
	i_LSM:= i_LSM ,
	i_LSH:= i_LSH ,
	i_RouteType:= i_RouteType,
	i_Time_LSH_on:= i_Time_LSH_on ,
	i_Time_LSM_on:= i_Time_LSM_on ,
	i_Time_LSM_off:= i_Time_LSM_off ,
	i_Time_LSL_off:= i_Time_LSL_off ,
	i_TimeDelay:= i_TimeDelay ,
	i_ModeControl_Q5:= ModeControl_Q5 ,
	i_StepBackPump:= StepBackPump ,
	q_P1=> q_P1 ,
	q_VA551=> q_VA551 ,
	q_VA11=> q_VA11 ,
	q_VA51=> q_VA51 ,
	q_Alarm_Empty_Q5=> q_Alarm_Empty_Q5 ,
	q_StepBackPump=> StepBackPump);

(*блок контроля и управления возвратом моющих средств*)
Return_Flow(
	i_AlarmPause:= (Step>=30),  (*в аварии или в паузе мойки или неготовности маршрута*)
	i_FS:= i_FS ,
	i_StepBackPump:= StepBackPump ,
	i_RouteType:= i_RouteType ,
	i_Current_VolumeFC11:= i_Current_VolumeFC11 ,
	i_TimeDelayRetPump:= i_TimeDelayRetPump ,
	i_TimeDelayRetFlow:= i_TimeDelayRetFlow ,
	i_TimeAlarmBackFlow:= i_TimeAlarmBackFlow ,
	q_BackPump=> q_BackPump ,
	q_AlarmBackFlow=> q_AlarmBackFlow ,
	q_EndReturn=>EndReturn  ,
      q_Return_OK=>Return_OK ,
	q_ZeroCount_FC11=> q_ZeroCount_FC11 ,
	q_FC11_start=> q_FC11_start );

(*блок контроля потока в танк возвратной воды Q4*)
Control_Q4(
	i_Start:= Start_Control_Q4 ,
	i_Block_Q4_in:= i_Block_Q4_in ,
	i_VA401:= q_VA401 ,
	i_VA541:= q_VA541 ,
	i_TimeDelay:= i_TimeDelay ,
	q_VA401=> q_VA401 ,
	q_VA541=> q_VA541);

T_Process();
T_Delay();
T_LSH_on (IN:=i_LSH,     PT:=DINT_TO_TIME(i_Time_LSH_on*1000));
T_LSM_on (IN:=i_LSM,     PT:=DINT_TO_TIME(i_Time_LSM_on*1000));
T_LSM_off(IN:=NOT i_LSM, PT:=DINT_TO_TIME(i_Time_LSM_off*1000));
T_LSL_off(IN:=NOT i_LSL, PT:=DINT_TO_TIME(i_Time_LSL_off*1000));
END_FUNCTION_BLOCK

(* POU Q4_Level, ST *)
FUNCTION_BLOCK Q4_Level (*блок контроля потока в танк возвратной воды Q4*)
VAR_INPUT
	i_Start                    : BOOL; (*запуск блока*)
	i_Block_Q4_in        : BOOL; (*блокировка подачи в Q4 - макс уровень и ph*)
	i_VA401                 : BOOL; (*клапан подачи в танк возвратной воды - вход от внешнего FB*)
	i_VA541                 : BOOL; (*клапан сброса в канализацию  - вход от внешнего FB*)
	i_TimeDelay           : DINT ; (*время задержки вкл/выкл клапанов и насосов*)
END_VAR

VAR_OUTPUT
	q_VA401               : BOOL; (*клапан подачи в танк возвратной воды*)
	q_VA541               : BOOL; (*клапан сброса в канализацию*)
END_VAR

VAR
	Step_Q4: INT;
	T_Delay: TON;
END_VAR
(*передача команд от внешнего FB на выход, если контроль Q4 выключен*)
q_VA401 := i_VA401;
q_VA541 := i_VA541;


     IF i_Start THEN
			        CASE Step_Q4 OF
			        0: (*возврат в Q4*)
			           q_VA401:= TRUE;
			           q_VA541:=TRUE; (*НО*)
			           T_Delay.PT:=T#3s;
			           T_Delay.IN:=i_Block_Q4_in;
			           IF T_Delay.Q THEN
			               T_Delay.IN:=FALSE;
			               Step_Q4:=1;
			           END_IF;
			        1: (*переключение*)
			           q_VA401:= TRUE;
			           T_Delay.PT:=DINT_TO_TIME(i_TimeDelay*1000);
			           T_Delay.IN:=TRUE;
			           IF T_Delay.Q THEN
			               T_Delay.IN:=FALSE;
			               Step_Q4:=2;
			           END_IF;
			        2: (*возврат в канализацию, в Q4 заблокировано*)
			           T_Delay.PT:=T#3s;
			           T_Delay.IN:=NOT i_Block_Q4_in;
			           IF T_Delay.Q THEN
			               T_Delay.IN:=FALSE;
			               Step_Q4:=3;
			           END_IF;
			        3: (*переключение*)
			           q_VA401:= TRUE;
			           T_Delay.PT:=DINT_TO_TIME(i_TimeDelay*1000);
			           T_Delay.IN:=TRUE;
			           IF T_Delay.Q THEN
			               T_Delay.IN:=FALSE;
			               Step_Q4:=0;
			           END_IF;
			        END_CASE;

     ELSE
               Step_Q4:=0;
               T_Delay.IN:=FALSE;

    END_IF;


T_Delay();
END_FUNCTION_BLOCK

(* POU Q5_Level, ST *)
FUNCTION_BLOCK Q5_Level (*блок поддержания уровня в циркуляционном баке во время мойки и при откачке*)
VAR_INPUT
	i_P1                       	: BOOL;
	i_VA551                 	: BOOL;
	i_VA11                   	: BOOL;
	i_VA51                   	: BOOL;
	i_LSL                     	: BOOL;      (*датчик уровня в циркуляционном баке*)
	i_LSM                   	: BOOL;      (*датчик уровня в циркуляционном баке*)
	i_LSH                    	: BOOL;      (*датчик уровня в циркуляционном баке*)
	i_RouteType           	: DINT ; (*тип маршрута 1 - емкостной,0 - замкнутый*)
	i_Time_LSH_on      	: DINT ; (*время задержки срабатывания датчика верх уровня цирк бака*)
	i_Time_LSM_on      	: DINT ; (*время задержки срабатывания датчика сред уровня цирк бака*)
	i_Time_LSM_off      	: DINT ; (*время задержки отключения датчика сред уровня цирк бака*)
	i_Time_LSL_off       	: DINT ; (*время задержки отключения датчика ниж уровня цирк бака*)
	i_TimeDelay            	: DINT ; (*время задержки вкл/выкл клапанов и насосов*)
	i_ModeControl_Q5   	: INT;    (*режим поддержания уровня: 0 - выкл, 1 - во время мойки через цирк бак, 2 - при промывке и вытесн через цирк бак*)
	i_StepBackPump   	: INT;
END_VAR

VAR_OUTPUT
	q_P1                     	: BOOL;
	q_VA551                	: BOOL;
	q_VA11                  	: BOOL;
	q_VA51                  	: BOOL;
	q_Alarm_Empty_Q5	: BOOL;(*авария опустошения цирк бака при работе на замкн маршруте*)
	q_StepBackPump   	: INT; (*задание режима работы возврата: 0 - отключено, 1 - старт возврата, 2 - пауза, 3 - докачка*)

END_VAR

VAR
	Step_Q5  AT %M*	: INT;
	T_LSL_off           	:TON;
	T_LSH_on           	:TON;
	T_LSM_on           	:TON;
	T_LSM_off           	:TON;
	T_Delay               	:TON;  (*служебный таймер*)
END_VAR
(*передача команд от внешнего FB на выход при выключенном контроле*)
q_P1      := i_P1;
q_VA551:= i_VA551;
q_VA11  := i_VA11;
q_VA51  := i_VA51;
q_StepBackPump:=i_StepBackPump;

CASE i_ModeControl_Q5 OF

0: (*контроль выключен*)
Step_Q5 := 0;
T_Delay.IN:=FALSE;

(*-------------------------------------------------------------------*)
1: (*контроль уровня во время мойки через цирк бак*)
   q_VA51:=TRUE;

		      CASE Step_Q5 OF
		      0: (*на среднем*)
		         q_P1:=TRUE;
		         q_StepBackPump:=1; (*включен возврат и контроль возврата*)
		         IF T_LSH_on.Q THEN
		            Step_Q5:=1;
		         ELSIF T_LSL_off.Q AND NOT i_LSM THEN
		            Step_Q5:=2;
		         END_IF;
		      1: (*на верхнем*)
		         q_P1:=TRUE;
		         q_StepBackPump:=2; (* пауза возврата*)
		         IF T_LSM_off.Q THEN
		            Step_Q5:=0;
		         END_IF;
		      2: (*на нижнем*)
		         q_StepBackPump:=1; (*включен возврат и контроль возврата*)
		         IF T_LSM_on.Q AND i_LSL THEN
		            Step_Q5:=0;
		         END_IF;
		         IF i_RouteType=0 THEN (*авария опустошения цирк бака при работе на замкн маршруте*)
		           q_Alarm_Empty_Q5:=TRUE;
		          END_IF;
		      END_CASE;

(*---------------------------------------------------------------------------*)
2: (*контроль уровня при промывке и вытесн через цирк бак*)
   q_P1:=TRUE;

				      CASE Step_Q5 OF
				      0: (*заполнение цирк бака*)
				         q_VA551:=TRUE;
				         q_VA11 :=TRUE;
				         IF T_LSM_on.Q THEN
				            Step_Q5:=1;
				         END_IF;
				      1: (*переключение*)
				         q_VA551:=TRUE;
				         q_VA51:=TRUE;
				         q_VA11:=TRUE;
				         T_Delay.PT:=DINT_TO_TIME(i_TimeDelay*1000);
				         T_Delay.IN:=TRUE;
				         IF T_Delay.Q THEN
				            T_Delay.IN:=FALSE;
				            Step_Q5:=2;
				         END_IF;
				      2: (*на среднем*)
				         q_VA551:=TRUE;
				         q_VA51:=TRUE;
				         IF T_LSH_on.Q THEN
				             Step_Q5:=3;
				         ELSIF T_LSL_off.Q AND NOT i_LSM THEN
				             Step_Q5:=4;
				         END_IF;
				      3: (*на верхнем*)
				         q_VA51:=TRUE;
				         IF T_LSM_off.Q THEN
				             Step_Q5:=2;
				         END_IF;
				      4: (*переключение*)
				         q_VA551:=TRUE;
				         q_VA51:=TRUE;
				         q_VA11:=TRUE;
				         T_Delay.PT:=DINT_TO_TIME(i_TimeDelay*1000);
				         T_Delay.IN:=TRUE;
				         IF T_Delay.Q THEN
				             T_Delay.IN:=FALSE;
				             Step_Q5:=2;
				         END_IF;
				      END_CASE;


END_CASE;

T_Delay();
T_LSH_on (IN:=i_LSH,     PT:=DINT_TO_TIME(i_Time_LSH_on*1000));
T_LSM_on (IN:=i_LSM,     PT:=DINT_TO_TIME(i_Time_LSM_on*1000));
T_LSM_off(IN:=NOT i_LSM, PT:=DINT_TO_TIME(i_Time_LSM_off*1000));
T_LSL_off(IN:=NOT i_LSL, PT:=DINT_TO_TIME(i_Time_LSL_off*1000));
END_FUNCTION_BLOCK

(* POU WashWater, ST *)
FUNCTION_BLOCK WashWater
VAR_INPUT
	i_Diag: BOOL;
	i_Pause: BOOL;
	i_Block_Q4_out  : BOOL; (*блокировка выпуска для полоскания из Q4  - мин уровень и ph*)
	i_Block_Q4_in: BOOL;	 (*блокировка подачи в Q4 - макс уровень и ph*)
	i_Ready_Route: BOOL; (*сигнал о готовности выбранного маршрута, если 0 - запрет старта процесса или в паузу *)
	i_type: INT;            (*тип мойки: 0-мойка водой, 1-терм дезинф*)

	i_FS: BOOL;       (*датчик протока на возврате*)
	i_LSL: BOOL;      (*датчик уровня в циркуляционном баке*)
	i_LSM: BOOL;      (*датчик уровня в циркуляционном баке*)
	i_LSH: BOOL;      (*датчик уровня в циркуляционном баке*)

	i_TE1: REAL;      (*температура на подаче*)
	i_TE2: REAL;      (*температура на возврате*)
	i_Current_VolumeFC1 : REAL;  (*текуший объем расходомера дезинфектанта*)
	i_Current_VolumeFC11: REAL;  (*текуший объем расходомера подачи*)

	i_TimeDelay           : DINT ; (*время задержки вкл/выкл клапанов и насосов*)
	i_Time_LSH_on         : DINT ; (*время задержки срабатывания датчика верх уровня цирк бака*)
	i_Time_LSM_on         : DINT ; (*время задержки срабатывания датчика сред уровня цирк бака*)
	i_Time_LSM_off        : DINT ; (*время задержки отключения датчика сред уровня цирк бака*)
	i_Time_LSL_off        : DINT ; (*время задержки отключения датчика ниж уровня цирк бака*)
	i_TimeProcess         : DINT ; (*время мойки*)
	i_TimeSwillWater      : DINT ; (*время промывки водой со сбросом в Q4*)
	i_TempProcess         : REAL ; (*температура мойки*)
	i_DeltaTempStartTime  : DINT ; (*перепад температуры для начала терм дезинфекции*)
	i_TempCool            : REAL ; (*температура охлаждения терм дезинфекции*)


	i_RouteType           : DINT ; (*тип маршрута 1 - емкостной,0 - замкнутый*)
	i_PumpCapacity        : DINT ; (*производительность подающего насоса *)
	i_TimeDelayRetPump    : DINT ; (*время задержки включения насоса возврата - объем подачи перед вкл*)
	i_TimeDelayRetFlow    : DINT ; (*время появления протока на возврате*)
	i_TimeAlarmBackFlow   : DINT ; (*время задержки аварии отсутсвия обратного протока*)
	i_VolumeDesinf        : DINT ; (*объем дезинфектанта*)
	i_Using_Q5          :DINT;       (*использование циркуляционного бака на мойках растворами и водой, 1 - использовать*)

    Step: INT;
END_VAR
VAR_OUTPUT
	q_VA541: BOOL;
	q_VA401: BOOL;
	q_VA11 : BOOL;
	q_VA551: BOOL;
	q_VA501: BOOL;
	q_VA51 : BOOL;
	q_VA511: BOOL;
	q_VA521: BOOL;
	q_VA531: BOOL;
	q_VE551: BOOL;
	q_P1   : BOOL;
	q_P12  : BOOL;
	q_Red  : BOOL;
	q_Yellow : BOOL;
	q_Green  : BOOL;
	q_Sirena : BOOL;
	q_BackPump: BOOL;
	q_Heating_VR1: BOOL;
	q_AlarmBackFlow:BOOL;  (* авария протока на возврате*)
	q_AlarmQ4: BOOL;       (*неготовность танка Q4, пауза процесса*)
	q_Alarm_Empty_Q5: BOOL;(*авария опустошения цирк бака при работе на замкн маршруте*)
	q_Vis_tim_Process:BOOL;
	q_FC1_start : BOOL;   (*старт подсчета импульсов дезинф*)
	q_FC11_start: BOOL;	  (*старт подсчета импульсов*)
	q_ZeroCount_FC1: BOOL; (*обнуление счетчика дезинф*)
	q_ZeroCount_FC11: BOOL; (*обнуление счетчика*)
	q_SP_P1 : REAL;
	q_SP_VR1: REAL;
	q_VisuMode: INT;
END_VAR

VAR

	Cool                    AT %M*: BOOL; (*во время термич дезинфекции было охлаждение*)
	PastPrev             AT %M*: INT;
	StepBackPump   AT %M*: INT; (*задание режима работы возврата: 0 - отключено, 1 - старт возврата, 2 - пауза, 3 - докачка*)
	Last_Time_min    AT %M*: DINT;  (*расчет оставшихся минут процесса*)
	Last_Time_sec    AT %M*: DINT;  (*расчет оставшихся секунд процесса*)

	EndReturn            :BOOL;  (* окончание докачки из маршрута*)
	Return_OK            :BOOL;  (* таймера отсчитали, идет возврат - норма*)
      Start_Control_Q4   :BOOL ;   (*старт процесса контроля потока в танк возвратной воды Q4 *)
	ModeControl_Q5   : INT;    (*режим поддержания уровня в цирк баке: 0 - выкл, 1 - во время мойки через цирк бак, 2 - при промывке и вытесн через цирк бак*)
	T_Delay   :TON;  (*служебный таймер*)
	T_LSL_off :TON;
	T_LSH_on  :TON;
	T_LSM_on  :TON;
	T_LSM_off :TON;
	T_Process :TON;
	Return_Flow : BackPump; (*блок контроля и управления возвратом моющих средств*)
	Control_Q4 :Q4_Level;   (*блок контроля потока в танк возвратной воды Q4*)
	Control_Q5 :Q5_Level;  (*блок поддержания уровня в циркуляционном баке во время мойки и при откачке*)
END_VAR
(*обнуление в начале скана*)
	q_VA541 := FALSE;  (*НО*)
	q_VA401 := FALSE;
	q_VA11  := FALSE;
	q_VA551 := FALSE;
	q_VA501 := FALSE;
	q_VA51  := FALSE;
	q_VA511 := FALSE;
	q_VA521 := FALSE;
	q_VA531 := FALSE;  (*НО*)
	q_VE551  := FALSE;
	q_P1 := FALSE;
	q_P12 := FALSE;
    q_Green :=FALSE;
    q_Yellow :=FALSE;
    q_Red:=FALSE;
    q_Sirena :=FALSE;
	q_BackPump := FALSE;
    q_Heating_VR1 := FALSE;
    q_AlarmBackFlow := FALSE;
    q_AlarmQ4:=FALSE;
    q_Alarm_Empty_Q5:=FALSE;
    q_Vis_tim_Process := FALSE;
	q_FC1_start  := FALSE;
	q_FC11_start := FALSE;
	q_ZeroCount_FC1  := FALSE;
	q_ZeroCount_FC11 := FALSE;
      Start_Control_Q4 := FALSE;
	q_SP_P1 :=0.0 ;
	q_SP_VR1 :=0.0 ;
      ModeControl_Q5 := 0;

(*выход в аварию*)
IF i_Diag   THEN
   IF Step=0 THEN
      PastPrev:=0;
   END_IF;
   Step:=30;
END_IF;

(*выход в паузу*)
IF i_Pause   THEN
   IF Step=0 THEN
      PastPrev:=0;
   END_IF;
   Step:=35;
END_IF;

(*выход в паузу по неготовности маршрута*)
IF NOT i_Ready_Route THEN
   IF Step=0 THEN
      PastPrev:=0;
   END_IF;
   Step:=36;
END_IF;

CASE Step OF
0: (*обнуление*)
  T_Delay.IN:=FALSE;
  T_Process.IN:=FALSE;
  q_ZeroCount_FC1:=TRUE;
  q_ZeroCount_FC11:=TRUE;
  Cool:=FALSE;

  StepBackPump := 0;
  Step:=1;

1: (*открытие клапанов, пуск насосов, подача в маршрут*)
  PastPrev:=Step;
  q_VA11:=TRUE;
  q_VA501:=TRUE;
  q_VA541:=TRUE; (*НО*)
  q_P1:=TRUE;
  q_SP_P1:=i_PumpCapacity;
  StepBackPump:=1; (*включен возврат и контроль возврата*)

  IF T_LSM_on.Q THEN
     Step:=2;
  END_IF;

  q_VisuMode:=2;

2: (*переключение*)
  PastPrev:=Step;
  q_VA11:=TRUE;
  q_VA51:=TRUE;
  q_VA501:=TRUE;
  q_VA541:=TRUE; (*НО*)
  q_P1:=TRUE;
  q_SP_P1:=i_PumpCapacity;
  StepBackPump:=1; (*включен возврат и контроль возврата*)


  T_Delay.PT:=DINT_TO_TIME(i_TimeDelay*1000);
  T_Delay.IN:=TRUE;
  IF T_Delay.Q THEN
     T_Delay.IN:=FALSE;
     Step:=3;
  END_IF;

  q_VisuMode:=2;


3: (*догрев*)
  PastPrev:=Step;
  q_VA541:=TRUE; (*НО*)
  q_VA501:=TRUE;
  q_Heating_VR1:=TRUE;
  q_SP_VR1 := i_TempProcess;
  q_SP_P1:=i_PumpCapacity;

  ModeControl_Q5 := 1; (*поддержание уровня в цирк баке во время мойки через цирк бак, контроль насоса Р1 и q_VA51*)


   IF i_type=0 AND i_TE1>=(i_TempProcess-1.0) THEN                      (*условие для мойки водой*)
      T_Process.PT:=DINT_TO_TIME(i_TimeProcess*60000);
      Step:=4;
   ELSIF i_type=1 AND i_TE2>=(i_TempProcess-i_DeltaTempStartTime) AND i_TE1>=(i_TempProcess-1.0) THEN (*условие для термической дезинфекции*)
      T_Process.PT:=DINT_TO_TIME(i_TimeProcess*60000);
      Step:=4;
   END_IF;

     q_VisuMode:=8;


4: (*отсчет времени*)
  PastPrev:=Step;
  q_VA541:=TRUE; (*НО*)
  q_VA501:=TRUE;
  q_Heating_VR1:=TRUE;
  q_SP_VR1 := i_TempProcess;
  q_SP_P1:=i_PumpCapacity;

  ModeControl_Q5 := 1; (*поддержание уровня в цирк баке во время мойки через цирк бак, контроль насоса Р1 и q_VA51*)

     (*расчет времени для визуализ*)
    q_Vis_tim_Process := TRUE; (*визуализация полей времени*)
    Last_Time_min := (TIME_TO_DINT(T_Process.PT-T_Process.ET))/60000 ;
    Last_Time_sec := (TIME_TO_DINT(T_Process.PT-T_Process.ET)/1000) - Last_Time_min * 60 ;

   T_Process.in:=TRUE;
   IF T_Process.Q THEN
      T_Process.in:=FALSE;
      Step:=5;
   END_IF;

  q_VisuMode:=3;

5: (*переключение*)
  PastPrev:=Step;
  q_VA51:=TRUE;
  q_VA501:=TRUE;
  q_VA401:=TRUE;
  q_VA541:=TRUE; (*НО*)
  q_P1:=TRUE;
  q_SP_P1:=i_PumpCapacity;
  StepBackPump:=1; (*включен возврат и контроль возврата*)

  T_Delay.PT:=DINT_TO_TIME(i_TimeDelay*1000);
  T_Delay.IN:=TRUE;
  IF T_Delay.Q THEN
     T_Delay.IN:=FALSE;
     Step:=6;
  END_IF;

  q_VisuMode:=4;

6:(*откачка из цирк бака*)
  PastPrev:=Step;
  q_VA51:=TRUE;
  q_P1:=TRUE;
  q_SP_P1:=i_PumpCapacity;
  StepBackPump:=1; (*включен возврат и контроль возврата*)

  Start_Control_Q4 := TRUE; (*контроль потока в танк возвратной воды Q4 *)

  IF (T_LSL_off.Q AND NOT i_LSM) THEN  (*циркуляционный бак пустой*)
      T_Delay.IN:=FALSE;
      IF  i_type=1 THEN
           IF i_TE2>i_TempCool THEN   (*если выбрана термич дезинфекция и темп высокая - на охлаждение*)
               Step:=7;
           ELSIF i_TE2<=i_TempCool THEN   (*если выбрана термич дезинфекция и темп низкая - докачка из маршрута*)
               Step:=9 ;
           END_IF;
      ELSE    (*если выбрана мойка водой*)
           IF i_TimeSwillWater = 0 THEN   (*если время ополаскивания со сбросом в Q4 равно 0 - докачка из маршрута*)
               Step:=9 ;
           ELSE
               T_Process.PT := DINT_TO_TIME(i_TimeSwillWater * 60000);
               T_Process.IN := FALSE ;
               Step:=7;
          END_IF;
      END_IF;
    END_IF;

  q_VisuMode:=4;

7: (*переключение на охлаждение / промывку со сбросом в Q4*)
  PastPrev:=Step;
  q_VA11:=TRUE;
  q_VA51:=TRUE;
  q_P1:=TRUE;
  q_SP_P1:=i_PumpCapacity;
  StepBackPump:=1; (*включен возврат и контроль возврата*)

  Start_Control_Q4 := TRUE; (*контроль потока в танк возвратной воды Q4 *)

  T_Delay.PT:=DINT_TO_TIME(i_TimeDelay*1000);
  T_Delay.IN:=TRUE;
  IF T_Delay.Q THEN
     T_Delay.IN:=FALSE;
     Step:=8;
  END_IF;

  q_VisuMode:=16;

8: (*охлаждение / промывка со сбросом в Q4*)
  PastPrev:=Step;
  q_VA11:=TRUE;
  q_P1:=TRUE;
  q_SP_P1:=i_PumpCapacity;
  StepBackPump:=1; (*включен возврат и контроль возврата*)
  Cool:=TRUE;           (*во время термич дезинфекции было охлаждение либо ополаскивание после мойки водой*)

  Start_Control_Q4 := TRUE; (*контроль потока в танк возвратной воды Q4 *)

      IF  i_type=1 THEN  (*охлаждение после термической дезинфекции*)
          IF i_TE2<=i_TempCool THEN (*достигли температуры охлаждения*)
              Step:=9;
          END_IF;
          q_VisuMode:=16;
      ELSE                      (*ополаскивание заданным временем после  мойки водой*)
          q_Vis_tim_Process := TRUE; (*визуализация полей времени*)
          Last_Time_min := (TIME_TO_DINT(T_Process.PT-T_Process.ET))/60000 ;
          Last_Time_sec := (TIME_TO_DINT(T_Process.PT-T_Process.ET)/1000) - Last_Time_min * 60 ;
          T_Process.in:=TRUE;
          IF T_Process.Q THEN
              T_Process.in:=FALSE;
              Step:=9;
          END_IF;
           q_VisuMode:=19;
    END_IF;


9: (*откачка из маршрута*)
  PastPrev:=Step;
  q_VA511:=TRUE;
  StepBackPump:=3; (*откачка из маршрута*)

(*задержка закрытия клапанов перед Р1*)
  T_Delay.PT:=DINT_TO_TIME(i_TimeDelay*1000); (*задержка закрытия клапана*)
  T_Delay.IN:=TRUE;
  q_VA11 := Cool AND  NOT T_Delay.Q ;
  q_VA51 :=  NOT Cool AND NOT T_Delay.Q;

  Start_Control_Q4 := TRUE; (*контроль потока в танк возвратной воды Q4 *)

  IF EndReturn THEN
     T_Delay.IN:= FALSE;
     StepBackPump := 0; (*выключить вовзрат и контроль возврата*)
     Step:=10;
  END_IF;

  q_VisuMode:=4;

10: (*выполнено*)
  q_VisuMode:=1;
  StepBackPump := 0; (*выключить вовзрат и контроль возврата*)




(*-----------------авария----------------*)
30: (*авария*)
       q_VisuMode:=11;
       q_Red:=TRUE;
       q_Sirena :=TRUE;
       T_Process.IN := FALSE; (*остановка таймера процесса*)
       IF AlarmReset AND (PastPrev=4 OR PastPrev=8)  THEN
          T_Process.PT := DINT_TO_TIME(Last_Time_min*60000 + Last_Time_sec*1000);  (*уставка для таймера  в случае выхода в аварию*)
          Step := PastPrev;
       ELSIF AlarmReset AND PastPrev<>4 AND PastPrev<>8 THEN
          Step := PastPrev;
       END_IF;

(*-----------------пауза----------------*)
35: (*пауза*)
       q_VisuMode:=12;
       q_Yellow:=TRUE;
       T_Process.IN := FALSE; (*остановка таймера процесса*)
       IF NOT i_Pause AND (PastPrev=4 OR PastPrev=8)  THEN
          T_Process.PT := DINT_TO_TIME(Last_Time_min*60000 + Last_Time_sec*1000);  (*уставка для таймера  в случае выхода в аварию*)
          Step := PastPrev;
       ELSIF NOT i_Pause AND PastPrev<>4 AND PastPrev<>8 THEN
          Step := PastPrev;
       END_IF;

(*-----------------пауза - не готов маршрут----------------*)
36: (*пауза*)
       q_VisuMode:=18;
       q_Yellow:=TRUE;
       T_Process.IN := FALSE; (*остановка таймера процесса*)
       IF i_Ready_Route AND (PastPrev=4 OR PastPrev=8)  THEN
          T_Process.PT := DINT_TO_TIME(Last_Time_min*60000 + Last_Time_sec*1000);  (*уставка для таймера  в случае выхода в аварию*)
          Step := PastPrev;
       ELSIF i_Ready_Route AND PastPrev<>4 AND PastPrev<>8THEN
          Step := PastPrev;
       END_IF;


 END_CASE;

(*блок поддержания уровня в циркуляционном баке во время мойки и при откачке*)
Control_Q5(
	i_P1:= q_P1,
	i_VA551:= q_VA551 ,
	i_VA11:= q_VA11 ,
	i_VA51:= q_VA51 ,
	i_LSL:= i_LSL ,
	i_LSM:= i_LSM ,
	i_LSH:= i_LSH ,
	i_RouteType:= i_RouteType,
	i_Time_LSH_on:= i_Time_LSH_on ,
	i_Time_LSM_on:= i_Time_LSM_on ,
	i_Time_LSM_off:= i_Time_LSM_off ,
	i_Time_LSL_off:= i_Time_LSL_off ,
	i_TimeDelay:= i_TimeDelay ,
	i_ModeControl_Q5:= ModeControl_Q5 ,
	i_StepBackPump:= StepBackPump ,
	q_P1=> q_P1 ,
	q_VA551=> q_VA551 ,
	q_VA11=> q_VA11 ,
	q_VA51=> q_VA51 ,
	q_Alarm_Empty_Q5=> q_Alarm_Empty_Q5 ,
	q_StepBackPump=> StepBackPump);

(*блок контроля и управления возвратом моющих средств*)
Return_Flow(
	i_AlarmPause:= (Step>=30),  (*в аварии или в паузе мойки или неготовности маршрута*)
	i_FS:= i_FS ,
	i_StepBackPump:= StepBackPump ,
	i_RouteType:= i_RouteType ,
	i_Current_VolumeFC11:= i_Current_VolumeFC11 ,
	i_TimeDelayRetPump:= i_TimeDelayRetPump ,
	i_TimeDelayRetFlow:= i_TimeDelayRetFlow ,
	i_TimeAlarmBackFlow:= i_TimeAlarmBackFlow ,
	q_BackPump=> q_BackPump ,
	q_AlarmBackFlow=> q_AlarmBackFlow ,
	q_EndReturn=>EndReturn  ,
      q_Return_OK=>Return_OK ,
	q_ZeroCount_FC11=> q_ZeroCount_FC11 ,
	q_FC11_start=> q_FC11_start );

(*блок контроля потока в танк возвратной воды Q4*)
Control_Q4(
	i_Start:= Start_Control_Q4 ,
	i_Block_Q4_in:= i_Block_Q4_in ,
	i_VA401:= q_VA401 ,
	i_VA541:= q_VA541 ,
	i_TimeDelay:= i_TimeDelay ,
	q_VA401=> q_VA401 ,
	q_VA541=> q_VA541);


T_Process();
T_Delay();
T_LSH_on (IN:=i_LSH,     PT:=DINT_TO_TIME(i_Time_LSH_on*1000));
T_LSM_on (IN:=i_LSM,     PT:=DINT_TO_TIME(i_Time_LSM_on*1000));
T_LSM_off(IN:=NOT i_LSM, PT:=DINT_TO_TIME(i_Time_LSM_off*1000));
T_LSL_off(IN:=NOT i_LSL, PT:=DINT_TO_TIME(i_Time_LSL_off*1000));
END_FUNCTION_BLOCK

(* POU ChemicDesinf, ST *)
FUNCTION_BLOCK ChemicDesinf  (*блок химической дезинфекции*)
VAR_INPUT
	i_Diag			: BOOL;
	i_Pause			: BOOL;
	i_Block_Q4_in	: BOOL;	 	(*блокировка подачи в Q4 - макс уровень и ph*)
	i_Alarm_LSmin	: BOOL;   	(*авария нижнего уровня в баке дезинфектанта*)
	i_Ready_Route	: BOOL; 	(*сигнал о готовности выбранного маршрута, если 0 - запрет старта процесса или в паузу *)

	i_FS	: BOOL;       	(*датчик протока на возврате*)
	i_LSL	: BOOL;      	(*датчик уровня в циркуляционном баке*)
	i_LSM	: BOOL;      	(*датчик уровня в циркуляционном баке*)
	i_LSH	: BOOL;      	(*датчик уровня в циркуляционном баке*)

	i_TE1					: REAL;      	(*температура на подаче*)
	i_TE2					: REAL;      	(*температура на возврате*)
	i_Current_VolumeFC1 	: REAL;  	(*текуший объем расходомера дезинфектанта*)
	i_Current_VolumeFC11	: REAL;  	(*текуший объем расходомера подачи*)

	i_TimeDelay           	: DINT ; (*время задержки вкл/выкл клапанов и насосов*)
	i_Time_LSH_on         	: DINT ; (*время задержки срабатывания датчика верх уровня цирк бака*)
	i_Time_LSM_on         : DINT ; (*время задержки срабатывания датчика сред уровня цирк бака*)
	i_Time_LSM_off        	: DINT ; (*время задержки отключения датчика сред уровня цирк бака*)
	i_Time_LSL_off        	: DINT ; (*время задержки отключения датчика ниж уровня цирк бака*)
	i_TimeProcess         	: DINT ; (*время мойки*)
	i_TimeSwill               	: DINT ; (*время ополаскивания чистой водой после дезинфекции, мин*)


	i_RouteType           		: DINT ; (*тип маршрута 1 - емкостной,0 - замкнутый*)
	i_PumpCapacity        	: DINT ; (*производительность подающего насоса *)
	i_TimeDelayRetPump    	: DINT ; (*время задержки включения насоса возврата - объем подачи перед вкл*)
	i_TimeDelayRetFlow    	: DINT ; (*время появления протока на возврате*)
	i_TimeAlarmBackFlow   	: DINT ; (*время задержки аварии отсутсвия обратного протока*)
	i_VolumeDesinf        		: DINT ; (*объем дезинфектанта*)

    Step: INT;
END_VAR
VAR_OUTPUT
	q_VA541	: BOOL;
	q_VA401	: BOOL;
	q_VA11 		: BOOL;
	q_VA551	: BOOL;
	q_VA501	: BOOL;
	q_VA51 		: BOOL;
	q_VA511	: BOOL;
	q_VA521	: BOOL;
	q_VA531	: BOOL;
	q_VE551	: BOOL;
	q_P1   		: BOOL;
	q_P12  		: BOOL;
	q_Red  		: BOOL;
	q_Yellow 	: BOOL;
	q_Green  	: BOOL;
	q_Sirena 	: BOOL;
	q_BackPump		: BOOL;
	q_Heating_VR1		: BOOL;
	q_AlarmBackFlow	: BOOL;  	(* авария протока на возврате*)
	q_AlarmQ4			: BOOL;       (*неготовность танка Q4, пауза процесса*)
	q_Alarm_Empty_Q5	: BOOL;		(*авария опустошения цирк бака при работе на замкн маршруте*)
	q_Vis_tim_Process	: BOOL;
	q_FC1_start 			: BOOL;   	(*старт подсчета импульсов дезинф*)
	q_FC11_start		: BOOL;	  	(*старт подсчета импульсов*)
	q_ZeroCount_FC1	: BOOL; 	(*обнуление счетчика дезинф*)
	q_ZeroCount_FC11	: BOOL; 	(*обнуление счетчика*)
	q_SP_P1 			: REAL;
	q_SP_VR1			: REAL;
	q_VisuMode			: INT;
END_VAR

VAR

	PastPrev             AT %M*: INT;
	StepBackPump   	AT %M*: INT; 	(*задание режима работы возврата: 0 - отключено, 1 - старт возврата, 2 - пауза, 3 - докачка*)
	Last_Time_min    AT %M*: DINT;  	(*расчет оставшихся минут процесса*)
	Last_Time_sec    AT %M*: DINT;  	(*расчет оставшихся секунд процесса*)

	EndReturn            	:BOOL;  	(* окончание докачки из маршрута*)
	Return_OK            	:BOOL;  	(* таймера отсчитали, идет возврат - норма*)
      Start_Control_Q4   	:BOOL ;   	(*старт процесса контроля потока в танк возвратной воды Q4 *)
	ModeControl_Q5   	: INT;    		(*режим поддержания уровня в цирк баке: 0 - выкл, 1 - во время мойки через цирк бак, 2 - при промывке и вытесн через цирк бак*)
	T_Delay   			:TON;  		(*служебный таймер*)
	T_LSL_off 			:TON;
	T_LSH_on  			:TON;
	T_LSM_on  			:TON;
	T_LSM_off 			:TON;
	T_Process 			:TON;
	Return_Flow 			: BackPump; (*блок контроля и управления возвратом моющих средств*)
	Control_Q4 			:Q4_Level;   	(*блок контроля потока в танк возвратной воды Q4*)
	Control_Q5 			:Q5_Level;  	(*блок поддержания уровня в циркуляционном баке во время мойки и при откачке*)
END_VAR
(*обнуление в начале скана*)
	q_VA541 := FALSE;  (*НО*)
	q_VA401 := FALSE;
	q_VA11  := FALSE;
	q_VA551 := FALSE;
	q_VA501 := FALSE;
	q_VA51  := FALSE;
	q_VA511 := FALSE;
	q_VA521 := FALSE;
	q_VA531 := FALSE;  (*НО*)
	q_VE551  := FALSE;
	q_P1 := FALSE;
	q_P12 := FALSE;
    q_Green :=FALSE;
    q_Yellow :=FALSE;
    q_Red:=FALSE;
    q_Sirena :=FALSE;
	q_BackPump := FALSE;
    q_Heating_VR1 := FALSE;
    q_AlarmBackFlow := FALSE;
    q_AlarmQ4:=FALSE;
    q_Alarm_Empty_Q5:=FALSE;
    q_Vis_tim_Process := FALSE;
	q_FC1_start  := FALSE;
	q_FC11_start := FALSE;
	q_ZeroCount_FC1  := FALSE;
	q_ZeroCount_FC11 := FALSE;
      Start_Control_Q4 := FALSE;
	q_SP_P1 :=0.0 ;
	q_SP_VR1 :=0.0 ;
      ModeControl_Q5 := 0;

(*выход в аварию*)
IF i_Diag   THEN
   IF Step=0 THEN
      PastPrev:=0;
   END_IF;
   Step:=30;
END_IF;

(*выход в паузу*)
IF i_Pause   THEN
   IF Step=0 THEN
      PastPrev:=0;
   END_IF;
   Step:=35;
END_IF;

(*выход в паузу по неготовности маршрута*)
IF NOT i_Ready_Route THEN
   IF Step=0 THEN
      PastPrev:=0;
   END_IF;
   Step:=36;
END_IF;

CASE Step OF
0: (*обнуление*)
  T_Delay.IN:=FALSE;
  T_Process.IN:=FALSE;
  q_ZeroCount_FC1:=TRUE;
  q_ZeroCount_FC11:=TRUE;

  StepBackPump := 0;
  Step:=1;

1: (*открытие клапанов, пуск насосов, подача в маршрут*)
  PastPrev:=Step;
  q_VA11:=TRUE;
  q_VA501:=TRUE;
  q_VA541:=TRUE; (*НО*)
  q_P1:=TRUE;
  q_SP_P1:=i_PumpCapacity;
  StepBackPump:=1; (*включен возврат и контроль возврата*)

  IF T_LSM_on.Q THEN  (*достигли средний уровень в цирк баке*)
     Step:=2;
  END_IF;

  q_VisuMode:=2;

2: (*переключение*)
  PastPrev:=Step;
  q_VA11:=TRUE;
  q_VA51:=TRUE;
  q_VA501:=TRUE;
  q_VA541:=TRUE; (*НО*)
  q_P1:=TRUE;
  q_SP_P1:=i_PumpCapacity;
  StepBackPump:=1; (*включен возврат и контроль возврата*)


  T_Delay.PT:=DINT_TO_TIME(i_TimeDelay*1000);
  T_Delay.IN:=TRUE;
  IF T_Delay.Q THEN
     T_Delay.IN:=FALSE;
     Step:=3;
  END_IF;

  q_VisuMode:=2;

3: (*подача дезинфектанта*)
  PastPrev:=Step;
  q_VA541:=TRUE; (*НО*)
  q_VA501:=TRUE;
  q_VE551:= TRUE ;
  q_P12  :=TRUE;
  q_FC1_start:=TRUE;
  q_SP_P1:=i_PumpCapacity;

  ModeControl_Q5 := 1; (*поддержание уровня в цирк баке во время мойки через цирк бак, контроль насоса Р1 и q_VA51*)

   IF i_Current_VolumeFC1>=i_VolumeDesinf THEN         (*условие для химической дезинфекции*)
      T_Process.PT:=DINT_TO_TIME(i_TimeProcess*60000);
      Step:=4;
   END_IF;

   IF i_Alarm_LSmin  THEN  (*мин уровень в баке концентрата - авария*)
      Step:=30;
   END_IF;

   q_VisuMode:=15;


4: (*отсчет времени*)
  PastPrev:=Step;
  q_VA51:=TRUE;
  q_VA541:=TRUE; (*НО*)
  q_VA501:=TRUE;
  q_SP_P1:=i_PumpCapacity;

  ModeControl_Q5 := 1; (*поддержание уровня в цирк баке во время мойки через цирк бак, контроль насоса Р1*)

     (*расчет времени для визуализ*)
    q_Vis_tim_Process := TRUE; (*визуализация полей времени*)
    Last_Time_min := (TIME_TO_DINT(T_Process.PT-T_Process.ET))/60000 ;
    Last_Time_sec := (TIME_TO_DINT(T_Process.PT-T_Process.ET)/1000) - Last_Time_min * 60 ;

   T_Process.in:=TRUE;
   IF T_Process.Q THEN
      T_Process.in:=FALSE;
      Step:=5;
   END_IF;

  q_VisuMode:=3;

5: (*переключение*)
  PastPrev:=Step;
  q_VA51:=TRUE;
  q_VA501:=TRUE;
  q_VA401:=TRUE;
  q_VA541:=TRUE; (*НО*)
  q_P1:=TRUE;
  q_SP_P1:=i_PumpCapacity;
  StepBackPump:=1; (*включен возврат и контроль возврата*)

  T_Delay.PT:=DINT_TO_TIME(i_TimeDelay*1000);
  T_Delay.IN:=TRUE;
  IF T_Delay.Q THEN
     T_Delay.IN:=FALSE;
     Step:=6;
  END_IF;

  q_VisuMode:=4;

6:(*откачка из цирк бака*)
  PastPrev:=Step;
  q_VA51:=TRUE;
  q_P1:=TRUE;
  q_SP_P1:=i_PumpCapacity;
  StepBackPump:=1; (*включен возврат и контроль возврата*)

  Start_Control_Q4 := TRUE; (*контроль потока в танк возвратной воды Q4 *)


    IF (T_LSL_off.Q AND NOT i_LSM) THEN  (*циркуляционный бак пустой*)
      StepBackPump:=3;
      IF i_TimeSwill = 0 THEN  (*если время промывки 0, то оставляем дезинфектант в маршруте - без промывки водой*)
         Step:=11 ;
      ELSE
         Step:=7 ;
      END_IF;
    END_IF;

  q_VisuMode:=4;

7: (*откачка из маршрута*)
  PastPrev:=Step;
  StepBackPump:=3; (*откачка из маршрута*)

  T_Delay.PT:=DINT_TO_TIME(i_TimeDelay*1000); (*задержка закрытия клапана*)
  T_Delay.IN:=TRUE;
  q_VA51:=NOT T_Delay.Q ;

  Start_Control_Q4 := TRUE; (*контроль потока в танк возвратной воды Q4 *)


      IF EndReturn  THEN (*докачали из маршрута*)
          T_Delay.IN:= FALSE;
         StepBackPump:=0; (*выключить возврат и контроль возврата*)
         Step:=8;
      END_IF;

  q_VisuMode:=4;

